// TwinCAT 3 PLC project mover_demo
// ProgramVersion: 3.1.4024.12
// libraries:
//   CmpBitmapPool, * (System)
//   Tc2_Standard, * (Beckhoff Automation GmbH)
//   Tc2_System, * (Beckhoff Automation GmbH)
//   Tc3_JsonXml, * (Beckhoff Automation GmbH)
//   Tc3_Module, * (Beckhoff Automation GmbH)
//   VisuDialogs, * (System)
// project tree:
//   DUTs/Helptec/ enLamp.TcDUT, enState.TcDUT, structAlarm.TcDUT, structButton.TcDUT
//   DUTs/ PieceType_e.TcTLEO, Mover_st.TcDUT, Piece_st.TcDUT
//   / GlobalTextList.TcGTLO, PlcTask.TcTTO, Visualization Manager.TcVMO (not stored), VISU_TASK.TcTTO (not stored)
//   GVLs/ CONST.TcGVL, GVL.TcGVL, HMI.TcGVL, IN.TcGVL, OUT.TcGVL, PERS.TcGVL, PRG.TcGVL, SIMU.TcGVL
//   POUs/00_MAIN/ MAIN.TcPOU, _05_FLAGS.TcPOU
//   POUs/10_HMI/FB%27s/ FB_BUTTON.TcPOU (not stored), FB_LampeBNI007F.TcPOU (not stored), FB_STATE.TcPOU (not stored)
//   POUs/10_HMI/ _10_HMI.TcPOU, _11_PAR_CHK.TcPOU, _14_STATE.TcPOU
//   POUs/20_AUTO/BuR SuperTrack com/ gMoverAxis.TcGVL, BR_PaletteCmd_t.TcDUT, BR_SectionCommand_t.TcDUT, PaletteCmd_bits_t.TcDUT, TC_to_BR_t.TcDUT, BR_to_TC_t.TcDUT, BR_TrackCommand_t.TcDUT
//   POUs/20_AUTO/FB%27s/ GetTick.TcPOU (not stored), getPercent.TcPOU (not stored)
//   POUs/20_AUTO/FB%27s/Vorlagen/ FB_ABL_VORLAGE.TcPOU (not stored), POU_AUT_VORLAGE.TcPOU (not stored), POU_ERR_VORLAGE.TcPOU (not stored), _01_MAIN.TcPOU (not stored)
//   POUs/20_AUTO/FileMan/ FB_FileMan.TcPOU, FB_ReadJSON.TcPOU, LoadFromMemory.TcPOU, SaveInMemory.TcPOU
//   POUs/20_AUTO/Mover/ ApproachScenario_e.TcTLEO, DistToTravel.TcPOU, FB_BasePieceHolder.TcPOU, FB_Group.TcPOU, FB_Mover.TcPOU, FB_MoverMan.TcPOU, FB_My_Piece.TcPOU, FB_Piece.TcPOU, FB_PieceHolderMover.TcPOU, FB_Position.TcPOU, FB_SimuMoverAxis.TcPOU, FB_SortMoverByPos.TcPOU, FB_PieceHolder.TcPOU, FB_StationMan.TcPOU, FB_Station.TcPOU, IProcessSampleMover.TcIO, ISimuMoverTimers.TcIO, IStation.TcIO, MoverDict.TcDUT, MoverDirection_e.TcTLEO, MoverState_e.TcTLEO, PiecePos_e.TcDUT, PieceState_e.TcDUT, Pos2D_t.TcDUT, ProcessExec_e.TcDUT, StationDict.TcDUT
//   POUs/20_AUTO/ST100/ F_GetPercent.TcPOU, ST100_Load_e.TcTLEO, FB_ABL_LOAD.TcPOU, FB_ABL_MODIFY.TcPOU, FB_ABL_UNLOAD.TcPOU, FB_AUT_ABSTRACT.TcPOU, FB_ABL_100.TcPOU, FB_AUT_LOAD.TcPOU, FB_AUT_MODIFY.TcPOU, FB_AUT_UNLOAD.TcPOU, ProcessExecution_e.TcTLEO, ST100_e.TcTLEO, ST100_Modify_e.TcTLEO, ST100_Unload_e.TcTLEO
//   POUs/20_AUTO/TOOL/ ASSERT.TcPOU, EqualApproximately.TcPOU, EqualDelta.TcPOU, EqualEssentially.TcPOU, IObject.TcIO, SortBubbleLREAL.TcPOU
//   POUs/20_AUTO/ _20_AUTO.TcPOU
//   VISUs/ Custom.TcIPO (not stored), VISU_main.TcVIS

CONFIGURATION mover_demo
    RESOURCE PLC ON TwinCAT3
        TASK PlcTask(INTERVAL := T#10ms, PRIORITY := 20);
        PROGRAM MAIN WITH PlcTask : MAIN;
        PROGRAM test WITH PlcTask : test;
    END_RESOURCE
END_CONFIGURATION

// ---- DUTs/Helptec/enLamp.TcDUT
{attribute 'qualified_only'}
{attribute 'strict'}
TYPE enLamp :
(
	Aus         := 2#0000,  //Aus
    Gruen       := 2#0001,  //Grün
    GruenB      := 2#1001,  //Grün blinkt
    Rot         := 2#0010,  //Rot
    RotB        := 2#1010,  //Rot blinkt
    Gelb        := 2#0011,  //Gelb
    GelbB       := 2#1011,  //Gelb blinkt
    Blau        := 2#0100,  //Blau 
    BlauB       := 2#1100,  //Blau blinkt
    Orange      := 2#0101,  //Orange
    OrangeB     := 2#1101,  //Orange blinkt
    Benutzer    := 2#0110,  //Benutzerdefiniert (Violet)
    BenutzerB   := 2#1110,  //Benutzerdefiniert blinkt (Violet)
    Weiss       := 2#0111,  //Weiss
    WeissB      := 2#1111   //Weiss blinkt
);
END_TYPE

// ---- DUTs/Helptec/enState.TcDUT
{attribute 'to_string'}
TYPE enState :
	//	MACHINE STATE
(
	StateOFF	,		(*0	OFF 		PLC STARTUP, EMERGENCY STOP	*)
	StateAIRon	,		(*1	AIR OK		AIRPRESSURE ON	 	*)
	StateENGIZED,		(*2	ENERGY OK	ENERGY/SECURITY CIRQUIT CLOSED	*)
	StateREF	,		(*3	HOMING		SYSTEM INITIAL RESET (HOMING AXIS ETC) *)
	StateMANU	,		(*4	MANUEL		MANUEL MODE (TEACH AXIS, MANEL MOVEMENT	*)
	StateINIT	,		(*5	INITIALISE	SYSTEM RESET 	*)
	StateREADY	,		(*6	READY		SYSTEM READY TO START	*)
	StateSTOP	,		(*7	STOP		SYSTEM STOPPED	*)
	StateALARM	,		(*8	ALARM		ALARM ACTIV	*)
	StateSTEP	,		(*9	STEP		STEP BY STEP MODE	*)
	StateEND	,		(*10 END		END MODE (FINISH ALL CYCLES	*)
	StateLEER	,		(*11 EMPTY		RUNNING TILL EMPTY STATE *)
	StateAUTO			(*12 RUN		RUNNING AUTOMATIC MODE	*)
);
END_TYPE

// ---- DUTs/Helptec/structAlarm.TcDUT
TYPE structAlarm :
STRUCT
	xAlarmIN	:	BOOL;	//Alarm Trigger
	xAlarmOFF	:	BOOL;	//Alarm übersteuert (wird nicht ausgelöst)
	xAlarmSAVE	:	BOOL;	//Alarm gespeichert (muss quittiert werden)
	xAlarmQUIT	:	BOOL;	//Alarm quittieren
	xAlarmOUT	:	BOOL;	//Alarm aktiv
	tAlarmVERZ	:	TIME;	//Alarmverzögerung
	sAlarmText	:	STRING;	//Alarmtext
	bAlarmNr	:	BYTE;	//Zusatztext #
END_STRUCT
END_TYPE

// ---- DUTs/Helptec/structButton.TcDUT
TYPE structButton :
STRUCT
	button	:	BOOL;	// BUTTON SIGNAL FROM HMI
	disable	:	BOOL;	// FORCE BUTTON INACTIV
	rtrig	:	BOOL;	// RISING EDGE
	ftrig	:	BOOL;	// FALLING EDGE
	press	:	BOOL;	// BUTTON PRESSED
	on		:	BOOL;	// FUNCTION ON (GREEN)
	error	:	BOOL;	// FUNCTION ERROR (RED)
END_STRUCT
END_TYPE

// ---- DUTs/PieceType_e.TcTLEO
{attribute 'qualified_only'}
{attribute 'strict'}
{attribute 'to_string'}
TYPE PieceType_e :
(
	long,
	short,
	_max
);
END_TYPE

// ---- DUTs/Mover_st.TcDUT
TYPE Mover_st :
STRUCT
	iStation	: INT;	// Number of the assigned station
	iPos		: INT;	// Current position
	pPiece		: POINTER TO Piece_st;	// Pointer to a pieces
END_STRUCT
END_TYPE

// ---- DUTs/Piece_st.TcDUT
TYPE Piece_st :
STRUCT
	iWorkingTimeMili	: INT;	// Time spent in a station, expressed in ms
	iWaitingTimeMili	: INT;	// Time spent out of any station, waiting to be proceed
	uiStartTimeMili		: UINT;	// Entering time in a station, expressed as task time
	UUID				: UDINT;	// Universal Unique ID
	eType				: PieceType_e;	// type of pieces
END_STRUCT
END_TYPE

// ---- POUs/20_AUTO/BuR SuperTrack com/BR_PaletteCmd_t.TcDUT
{attribute 'pack_mode=1'}
TYPE BR_PaletteCmd_t :
STRUCT
    cmd        : PaletteCmd_bits_t;
    nextTarget : USINT;
    offset     : ARRAY[0..2] OF USINT;
END_STRUCT
END_TYPE

// ---- POUs/20_AUTO/BuR SuperTrack com/BR_SectionCommand_t.TcDUT
{attribute 'pack_mode=1'}
TYPE BR_SectionCommand_t :
STRUCT
    enable : BIT;
END_STRUCT
END_TYPE

// ---- POUs/20_AUTO/BuR SuperTrack com/PaletteCmd_bits_t.TcDUT
TYPE PaletteCmd_bits_t :
STRUCT
    releaseToTargetOffset : BIT;
    direction             : BIT;
END_STRUCT
END_TYPE

// ---- POUs/20_AUTO/BuR SuperTrack com/TC_to_BR_t.TcDUT
{attribute 'pack_mode=1'}
TYPE TC_to_BR_t :
STRUCT
    trackCmd   : BR_TrackCommand_t;
    paletteNum : USINT;

    sectionCmd : BR_SectionCommand_t;

    missingPaletteIDs : ARRAY[0..20] OF USINT;

    palettesCmd : ARRAY[0..40] OF BR_PaletteCmd_t;

END_STRUCT
END_TYPE

// ---- POUs/20_AUTO/BuR SuperTrack com/BR_to_TC_t.TcDUT
{attribute 'pack_mode=1'}
TYPE BR_to_TC_t :
STRUCT
END_STRUCT
END_TYPE

// ---- POUs/20_AUTO/BuR SuperTrack com/BR_TrackCommand_t.TcDUT
{attribute 'pack_mode=1'}
TYPE BR_TrackCommand_t :
STRUCT
    enableAllSections        : BIT;
    releasePaletteAtTarget_1 : BIT;
    ApplyPaletteNumber       : BIT;
END_STRUCT
END_TYPE

// ---- POUs/20_AUTO/Mover/ApproachScenario_e.TcTLEO
{attribute 'qualified_only'}
{attribute 'strict'}
{attribute 'to_string'}
TYPE
ApproachScenario_e :
(
    WaitOnFinishedProcess,
    WaitOnFreeStation,
    DoNotWait,
    WaitOnPrevProcess,
    WaitOnExternalTrigger,
    _MAX
);
END_TYPE

// ---- POUs/20_AUTO/Mover/MoverDict.TcDUT
// Get information from a mover using this structure
TYPE MoverDict :
STRUCT
    MoverNum : INT;
    MoverPos : LREAL;
END_STRUCT
END_TYPE

// ---- POUs/20_AUTO/Mover/MoverDirection_e.TcTLEO
{attribute 'qualified_only'}
{attribute 'strict'}
TYPE MoverDirection_e :
(
	Farward,
	Reverse
);
END_TYPE

// ---- POUs/20_AUTO/Mover/MoverState_e.TcTLEO
{attribute 'qualified_only'}
{attribute 'strict'}
{attribute 'to_string'}
TYPE
MoverState_e :
(
    OperationDone,           // The operation on the mover is done, a new station needs to be given
    WaitOnNextStation,       // wait on the next station to be ready. The waiting depend on the scenario of the next station
    WaitLeaveCurrentStation, // If we are bind with the track system, we will be sure that we have actualy leaved the curent station
    MovingToStation,         // the mover is moving or try to move to the next station
    InStationPos,            // The mover is currently AT the station position (aka target pos.), waiting on the process TO begin
    InOperation,             // The attached process of the mover is running. The mover is not able to move
    PerformRelativeMove,     // Moving the mover when already in operation, go to WaitRelativeMoveEnd when mover actually moving
    WaitRelativeMoveEnd,     // Wait on the At_pos flag
    _MAX
);
END_TYPE

// ---- POUs/20_AUTO/Mover/PiecePos_e.TcDUT
{attribute 'qualified_only'}
{attribute 'strict'}
TYPE PiecePos_e :
(
    Assembly_left  := 0,
    Assembly_right := 1,
    Test_left      := 2,
    Test_right     := 3,
    _max           := 4
);
END_TYPE

// ---- POUs/20_AUTO/Mover/PieceState_e.TcDUT
{attribute 'qualified_only'}
{attribute 'strict'}
{attribute 'to_string'}
/// Piece status
TYPE PieceState_e :
(
    bad     := -1,
    good    := 0,
    working := 1 // a station works on a piece or has not finished its process
);
END_TYPE

// ---- POUs/20_AUTO/Mover/Pos2D_t.TcDUT
TYPE
Pos2D_t :
STRUCT
    x : DINT;
    y : DINT;
END_STRUCT
END_TYPE

// ---- POUs/20_AUTO/Mover/ProcessExec_e.TcDUT
{attribute 'qualified_only'}
{attribute 'strict'}
{attribute 'to_string'}
TYPE ProcessExec_e :
(
	StartImmediately,
	StartSynchronize,
	_MAX
);
END_TYPE

// ---- POUs/20_AUTO/Mover/StationDict.TcDUT
// Get information from a mover using this structure
TYPE StationDict :
STRUCT
    StationNum : INT;
    StationPos : LREAL;
END_STRUCT
END_TYPE

// ---- POUs/20_AUTO/ST100/ST100_Load_e.TcTLEO
{attribute 'qualified_only'}
{attribute 'strict'}
TYPE
ST100_Load_e :
(
    RESET := 0,         // Reset
    INIT := 100,        // Initialisieren 
    READY := 999,       // READY to Start, Init Done 
    START := 1000,      // Start Zyklisch
    MOVER_FREE_OP,      // Ab here, operation without mover can be done
    proceedOperation_1, // proceed to some operation
    waitOnMover,        // wait until the mover is there
    MOVER_NEEDED_OP,    // Ab here, a mover in position is needed to perform the action
    proceedOperation_2, // proceed to some operation
    SYNC_MOVER_LEAVE,   // MoverMan need to take the mover
    DONE := 8000,       // Ablauf beendet 
    ERROR := 9000,      // Fehler 
    _max
);
END_TYPE

// ---- POUs/20_AUTO/ST100/ProcessExecution_e.TcTLEO
{attribute 'qualified_only'}
{attribute 'strict'}
{attribute 'to_string'}
TYPE ProcessExecution_e :
(
	ExecuteImmediately,
	ExecuteWithPrevious,
	_MAX
);
END_TYPE

// ---- POUs/20_AUTO/ST100/ST100_e.TcTLEO
{attribute 'qualified_only'}
{attribute 'strict'}
{attribute 'to_string'}
TYPE
ST100_e :
(
    RESET := 0,         // Reset
    INIT := 100,        // Initialisieren 
    READY := 999,       // READY to Start, Init Done 
    START := 1000,      // Start Zyklisch
    MOVER_FREE_OP,      // Ab here, operation without mover can be done
    proceedOperation_1, //proceed to some operation
    waitOnMover,        // wait until the mover is there
    MOVER_NEEDED_OP,    // Ab here, a mover in position is needed to perform the action
    proceedOperation_2, //proceed to some operation
    DONE := 8000,       // Ablauf beendet 
    ERROR := 9000,      // Fehler 
    _max
);
END_TYPE

// ---- POUs/20_AUTO/ST100/ST100_Modify_e.TcTLEO
{attribute 'qualified_only'}
{attribute 'strict'}
TYPE ST100_Modify_e :
(
    RESET := 0,         // Reset
    INIT := 100,        // Initialisieren 
    READY := 999,       // READY to Start, Init Done 
    START := 1000,      // Start Zyklisch
    MOVER_FREE_OP,      // Ab here, operation without mover can be done
    waitOnMover,        // wait until the mover is there
    MOVER_NEEDED_OP,    // Ab here, a mover in position is needed to perform the action
    proceedOperation_1, //proceed to some operation
    proceedOperation_2, //proceed to some operation
    SYNC_MOVER_LEAVE,   // MoverMan need to take the mover
    DONE := 8000,       // Ablauf beendet 
    ERROR := 9000,      // Fehler 
    _max
);
END_TYPE

// ---- POUs/20_AUTO/ST100/ST100_Unload_e.TcTLEO
{attribute 'qualified_only'}
{attribute 'strict'}
TYPE ST100_Unload_e :
(
    RESET := 0,         // Reset
    INIT := 100,        // Initialisieren 
    READY := 999,       // READY to Start, Init Done 
    START := 1000,      // Start Zyklisch
    waitOnMover,        // wait until the mover is there
    MOVER_NEEDED_OP,    // Ab here, a mover in position is needed to perform the action
    proceedOperation_1, //proceed to some operation
    SYNC_MOVER_LEAVE,   // MoverMan need to take the mover
    MOVER_FREE_OP,      // Ab here, operation without mover can be done
    proceedOperation_2, //proceed to some operation
    DONE := 8000,       // Ablauf beendet 
    ERROR := 9000,      // Fehler 
    _max
);
END_TYPE

// ---- GVLs/CONST.TcGVL
{attribute 'qualified_only' := ''}
VAR_GLOBAL CONSTANT
    (*******************************************************************)
    (* Globale KONSTANTEN *)
    (*******************************************************************)

    USE_SIMULATION  : BOOL := TRUE;
    BIND_WITH_TRACK : BOOL := FALSE;

    STATION_NUMBER        : INT   := 18;
    MAX_GROUP             : INT   := 6;
    MAX_STATION_PER_GROUP : INT   := 8;
    RECIPE_NUMBER         : INT   := 4;
    MAX_TRACK_LENGTH      : LREAL := 10000;
    MAX_MOVER_SIZE        : LREAL := 200.0;

    MOVER_NUMBER : INT := 18;

    MAX_TRACK_OFFSET_LIST  : INT := 10;
    MAX_RECIPE_PER_STATION : INT := 10;
END_VAR

// ---- GVLs/GVL.TcGVL
{attribute 'qualified_only'}
VAR_GLOBAL
    (*******************************************************************)
    (* Allgemeine Globale Variablen *)
    (*******************************************************************)
    (******* FREIGABEN *********)
    //ST01
    xFG_ST01akVZ : BOOL; // Vereinzelung Teil anwesend
    xFG_ST01akWT : BOOL; // WT anwesend
    //ST02
    xFG_ST02akWT : BOOL; // WT anwesend

END_VAR

// ---- GVLs/HMI.TcGVL
{attribute 'qualified_only'}
VAR_GLOBAL
(*******************************************************************)
(* Globale HMI Variablen *)
(*******************************************************************)
	xImmer0	: 	BOOL := FALSE;	//ALLWAYS FALSE
	xImmer1	: 	BOOL := TRUE;	//ALLWAYS TRUE

(*******************************************************************)
(* Flags *)
(*******************************************************************)
	enState		:	enState;	//SYSTEM STATUS
	xInitDone	:	BOOL;		//SYSTEM INITIALIZED
	xRefDone	:	BOOL;		//Axis REF
	xAlarm		:	BOOL;		//ALARM AKTIV
	xMessage	:	BOOL;		//MELDUNG AKTIV
	xWait		:	BOOL;		//ALLE FBs warten
	xAIRon		:	BOOL;		//Luftdruck IO
	xSPC		:	BOOL;		//SPC angewählt

(*******************************************************************)
(* Buttons *)
(*******************************************************************)
	//Control
	btArMain	: ARRAY[0..20] OF structButton;	(*	
													0: AUTO
													1: STEP
													2: END
													3: MANU
													4: INIT
													5: STOP
													6: LEER
													7: QUIT
													8: RESET TEMP COUNTER
													9: START
													10: ...
												*)
	//Manuel Station 1
	btArManu01	: ARRAY[0..10] OF structButton;	(*	
													0: Zyklus	
													1: 101.01
													2: 101.02
													3: 101.03
													*)
	//Manuel Station 2
	btArManu02	: ARRAY[0..10] OF structButton;(*	
													0: Zyklus	
													1: 
													*)
	//Manuel Station 3
	btArManu03	: ARRAY[0..10] OF structButton;(*	
													0: Zyklus	
													1: 
													*)
	//Manuel Station 4
	btArManu04	: ARRAY[0..10] OF structButton;	(*	
													0: Zyklus	
													1: 
													*)
	//Manuel Station 5
	btArManu05	: ARRAY[0..10] OF structButton;(*	
													0: Zyklus	
													1: 
													*)
	//Manuel Station 6
	btArManu06	: ARRAY[0..10] OF structButton;(*	
													0: Zyklus	
													1: 
													*)
	//Manuel Station 7
	btArManu07	: ARRAY[0..10] OF structButton;(*	
													0: Zyklus	
													1: 
													*)
	//Manuel Station 8
	btArManu08	: ARRAY[0..10] OF structButton;(*	
													0: Zyklus	
													1: 
													*)
	//Manuel Station 9
	btArManu09	: ARRAY[0..10] OF structButton;(*	
													0: Zyklus	
													1: 
													*)
	//Manuel Station 10
	btArManu10	: ARRAY[0..10] OF structButton;(*	
													0: Zyklus	
													1: 
													*) 

(*******************************************************************)
(* ALARME  *)
(*******************************************************************)				
	strArALARM : ARRAY [1..100] OF structAlarm;	
	strArMSG : ARRAY [1..100] OF structAlarm;
	xArAlarmHMI : ARRAY [1..9999] OF BOOL;
	
(*******************************************************************)
(* ANZEIGE - Werte *)
(*******************************************************************)

(*******************************************************************)
(* Cycle Time [STATION]*)
(*******************************************************************)
	dwArStartTime	: 	ARRAY[0..10] OF DWORD;
	dwArCycleTime	: 	ARRAY[0..10] OF DWORD;
	
(*******************************************************************)
(* Diverses *)
(*******************************************************************)
	xWriteALlog: BOOL;	//Alarmlog schreiben in File
END_VAR

// ---- GVLs/IN.TcGVL
{attribute 'qualified_only'}
VAR_GLOBAL
(*******************************************************************)
(* EINGÄNGE *)
(*******************************************************************)
	(* Modul *)
	//-EL#
//	I000_24VDC			AT %IX0.0		:	BOOL;			//Überwachung +24VDC
//	I001_				AT %IX0.1		:	BOOL;			//
//	I002_				AT %IX0.2		:	BOOL;			//    
//	I003_		    	AT %IX0.3		:	BOOL;			//	
//	I004_				AT %IX0.4		:	BOOL;			//Reserve
//	I005_				AT %IX0.5		:	BOOL;			//Reserve
//	I006_				AT %IX0.6		:	BOOL;			//Reserve    
//	I007_				AT %IX0.7		:	BOOL;			//Reserve
//	
//	I010_				AT %IX1.0		:	BOOL;			//Taktsignal Presse
//	I011_				AT %IX1.1		:	BOOL;			//Presse Bereit
//	I012_				AT %IX1.2		:	BOOL;			//Reserve Presse
//	I013_				AT %IX1.3		:	BOOL;			//Reserve Presse
//	I014_				AT %IX1.4		:	BOOL;			//Reserve
//	I015_				AT %IX1.5		:	BOOL;			//Reserve
//	I016_				AT %IX1.6		:	BOOL;			//Reserve
//	I017_				AT %IX1.7		:	BOOL;			//Reserve
//	
//	
//	(* IO-Link Boxen *)
//(*******************************************************************)
//	//-5001
//	(*Beispiel 	ST01 	Stopper Mono (nur GS), Greifer Mono, 
//						Vereinzelung Bi, AK WT, AK Teil, STAU WF
//	*)
//	IB5001				AT %IB5001			:	BYTE;			//Input Byte Box 1
//	I101_01_GS			AT %IX5001.0		:	BOOL;			//Stopper GS
//	I101_02_UH			AT %IX5001.1		:	BOOL;			//Greifer GS
//	I101_02_AS			AT %IX5001.2		:	BOOL;			//Greifer AS
//	I101_03_GS			AT %IX5001.3		:	BOOL;			//Vereinzelung GS
//	I101_03_AS			AT %IX5001.4		:	BOOL;			//Vereinzelung AS
//	I101_WT				AT %IX5001.5		:	BOOL;			//AK WT	
//	I101_AK				AT %IX5001.6		:	BOOL;			//AK Teil
//	I101_STAU			AT %IX5001.7		:	BOOL;			//Stau Zuführung
//	
//	//-5002
//	(*Beispiel 	ST02 	Stopper Mono (nur GS), Indexierer Mono, 
//						Presse Mono, AK WT, AK Teil
//	*)
//	IB5002				AT %IB5002			:	BYTE;			//Input Byte Box 2
//	I102_01_GS			AT %IX5002.0		:	BOOL;			//Stopper GS
//	I102_02_GS			AT %IX5002.1		:	BOOL;			//Index GS
//	I102_02_AS			AT %IX5002.2		:	BOOL;			//Index AS
//	I102_03_GS			AT %IX5002.3		:	BOOL;			//Pressen GS
//	I102_03_AS			AT %IX5002.4		:	BOOL;			//Pressen AS
//	I102_WT				AT %IX5002.5		:	BOOL;			//AK WT	
//	I102_AK				AT %IX5002.6		:	BOOL;			//AK Teil
//	I102_STAU			AT %IX5002.7		:	BOOL;			//
//	(*
//	IB5001				AT %IB5001			:	BYTE;			//Input Byte Box 1
//	I5001_0_			AT %IX5001.0		:	BOOL;			//
//	I5001_1_			AT %IX5001.1		:	BOOL;			//
//	I5001_2_			AT %IX5001.2		:	BOOL;			//
//	I5001_3_			AT %IX5001.3		:	BOOL;			//
//	I5001_4_			AT %IX5001.4		:	BOOL;			//
//	I5001_5_			AT %IX5001.5		:	BOOL;			//	
//	I5001_6_			AT %IX5001.6		:	BOOL;			//
//	I5001_7_			AT %IX5001.7		:	BOOL;			//
//	
//	//-5002
//	IB5002				AT %IB5002			:	BYTE;			//Input Byte Box 2
//	I5002_0_			AT %IX5002.0		:	BOOL;			//
//	I5002_1_			AT %IX5002.1		:	BOOL;			//
//	I5002_2_			AT %IX5002.2		:	BOOL;			//
//	I5002_3_			AT %IX5002.3		:	BOOL;			//
//	I5002_4_			AT %IX5002.4		:	BOOL;			//
//	I5002_5_			AT %IX5002.5		:	BOOL;			//	
//	I5002_6_			AT %IX5002.6		:	BOOL;			//
//	I5002_7_			AT %IX5002.7		:	BOOL;			//
//	*)
//	//-5003
//	IB5003				AT %IB5003			:	BYTE;			//Input Byte Box 3
//	I5003_0_			AT %IX5003.0		:	BOOL;			//
//	I5003_1_			AT %IX5003.1		:	BOOL;			//
//	I5003_2_			AT %IX5003.2		:	BOOL;			//
//	I5003_3_			AT %IX5003.3		:	BOOL;			//
//	I5003_4_			AT %IX5003.4		:	BOOL;			//
//	I5003_5_			AT %IX5003.5		:	BOOL;			//	
//	I5003_6_			AT %IX5003.6		:	BOOL;			//
//	I5003_7_			AT %IX5003.7		:	BOOL;			//
//	
//	//-5004
//	IB5004				AT %IB5004			:	BYTE;			//Input Byte Box 4
//	I5004_0_			AT %IX5004.0		:	BOOL;			//
//	I5004_1_			AT %IX5004.1		:	BOOL;			//
//	I5004_2_			AT %IX5004.2		:	BOOL;			//
//	I5004_3_			AT %IX5004.3		:	BOOL;			//
//	I5004_4_			AT %IX5004.4		:	BOOL;			//
//	I5004_5_			AT %IX5004.5		:	BOOL;			//	
//	I5004_6_			AT %IX5004.6		:	BOOL;			//
//	I5004_7_			AT %IX5004.7		:	BOOL;			//
//	
//	//-5005
//	IB5005				AT %IB5005			:	BYTE;			//Input Byte Box 5
//	I5005_0_			AT %IX5005.0		:	BOOL;			//
//	I5005_1_			AT %IX5005.1		:	BOOL;			//
//	I5005_2_			AT %IX5005.2		:	BOOL;			//
//	I5005_3_			AT %IX5005.3		:	BOOL;			//
//	I5005_4_			AT %IX5005.4		:	BOOL;			//
//	I5005_5_			AT %IX5005.5		:	BOOL;			//	
//	I5005_6_			AT %IX5005.6		:	BOOL;			//
//	I5005_7_			AT %IX5005.7		:	BOOL;			//
//	
//	//-5006
//	IB5006				AT %IB5006			:	BYTE;			//Input Byte Box 6
//	I5006_0_			AT %IX5006.0		:	BOOL;			//
//	I5006_1_			AT %IX5006.1		:	BOOL;			//
//	I5006_2_			AT %IX5006.2		:	BOOL;			//
//	I5006_3_			AT %IX5006.3		:	BOOL;			//
//	I5006_4_			AT %IX5006.4		:	BOOL;			//
//	I5006_5_			AT %IX5006.5		:	BOOL;			//	
//	I5006_6_			AT %IX5006.6		:	BOOL;			//
//	I5006_7_			AT %IX5006.7		:	BOOL;			//
//	
//	//-5007
//	IB5007				AT %IB5007			:	BYTE;			//Input Byte Box 7
//	I5007_0_			AT %IX5007.0		:	BOOL;			//
//	I5007_1_			AT %IX5007.1		:	BOOL;			//
//	I5007_2_			AT %IX5007.2		:	BOOL;			//
//	I5007_3_			AT %IX5007.3		:	BOOL;			//
//	I5007_4_			AT %IX5007.4		:	BOOL;			//
//	I5007_5_			AT %IX5007.5		:	BOOL;			//	
//	I5007_6_			AT %IX5007.6		:	BOOL;			//
//	I5007_7_			AT %IX5007.7		:	BOOL;			//
//	
//	//-5008
//	IB5008				AT %IB5008			:	BYTE;			//Input Byte Box 8
//	I5008_0_			AT %IX5008.0		:	BOOL;			//
//	I5008_1_			AT %IX5008.1		:	BOOL;			//
//	I5008_2_			AT %IX5008.2		:	BOOL;			//
//	I5008_3_			AT %IX5008.3		:	BOOL;			//
//	I5008_4_			AT %IX5008.4		:	BOOL;			//
//	I5008_5_			AT %IX5008.5		:	BOOL;			//	
//	I5008_6_			AT %IX5008.6		:	BOOL;			//
//	I5008_7_			AT %IX5008.7		:	BOOL;			//
//	
//	//-5009
//	IB5009				AT %IB5009			:	BYTE;			//Input Byte Box 9
//	I5009_0_			AT %IX5009.0		:	BOOL;			//
//	I5009_1_			AT %IX5009.1		:	BOOL;			//
//	I5009_2_			AT %IX5009.2		:	BOOL;			//
//	I5009_3_			AT %IX5009.3		:	BOOL;			//
//	I5009_4_			AT %IX5009.4		:	BOOL;			//
//	I5009_5_			AT %IX5009.5		:	BOOL;			//	
//	I5009_6_			AT %IX5009.6		:	BOOL;			//
//	I5009_7_			AT %IX5009.7		:	BOOL;			//
//	
//	//-5010
//	IB5010				AT %IB5010			:	BYTE;			//Input Byte Box 10
//	I5010_0_			AT %IX5010.0		:	BOOL;			//
//	I5010_1_			AT %IX5010.1		:	BOOL;			//
//	I5010_2_			AT %IX5010.2		:	BOOL;			//
//	I5010_3_			AT %IX5010.3		:	BOOL;			//
//	I5010_4_			AT %IX5010.4		:	BOOL;			//
//	I5010_5_			AT %IX5010.5		:	BOOL;			//	
//	I5010_6_			AT %IX5010.6		:	BOOL;			//
//	I5010_7_			AT %IX5010.7		:	BOOL;			//
	
END_VAR

// ---- GVLs/OUT.TcGVL
{attribute 'qualified_only'}
VAR_GLOBAL
(*******************************************************************)
(* AUSGÄNGE *)
(*******************************************************************)
	(* Modul *)	
	//-EL#
//	Q000_LAMP_NRJ		AT %QX0.0		:	BOOL;			//Lampe Energie
//	Q001_TuerVer		AT %QX0.1		:	BOOL;			//Türen verriegelt
//	Q002_				AT %QX0.2		:	BOOL;			//
//	Q003_				AT %QX0.3		:	BOOL;			//Reserve
//	Q004_WF_FG			AT %QX0.4		:	BOOL;			//ST01 Freigabe WF 
//	Q005_				AT %QX0.5		:	BOOL;			//Reserve
//	Q006_				AT %QX0.6		:	BOOL;			//
//	Q007_				AT %QX0.7		:	BOOL;			//
//	
//	Q010_				AT %QX1.0		:	BOOL;			//
//	Q011_				AT %QX1.1		:	BOOL;			//
//	Q012_				AT %QX1.2		:	BOOL;			//Reserve
//	Q013_				AT %QX1.3		:	BOOL;			//Reserve
//	Q014_				AT %QX1.4		:	BOOL;			//Reserve
//	Q015_				AT %QX1.5		:	BOOL;			//Reserve
//	Q016_				AT %QX1.6		:	BOOL;			//Reserve
//	Q017_				AT %QX1.7		:	BOOL;			//Reserve
//			
//
//	(* IO-Link  *)
//(*******************************************************************)
//	(* Lampe *)
//	QW194A3				AT%Q*			:	WORD;			//Signallampe1
//	QW194A6				AT%Q*			: 	WORD;			//Signallampe2
//	
//	Q194A3_SycStart		AT %Q*			:	BOOL;			//Syscstart 194A3
//	Q194A6_SycStart		AT %Q*			:	BOOL;			//Syscstart 194A6	
//	Q194A3_SycImp		AT %Q*			:	BOOL;			//SyscImp 194A3
//	Q194A6_SycImp		AT %Q*			:	BOOL;			//SyscImp 194A6		
//	
//	(* Boxen *)
//	(*Beispiel 	ST01 Stopper Mono, Greifer Mono, Vereinzelung Bi,
//				ST02 Stopper Mono, Indexierer Mono, Presse Mono
//	*)
//	Q101_01_AS			AT	%QX2000.0	:	BOOL;			//101.01 Stopper
//	Q200A1_1_12			AT	%QX2000.1	:	BOOL;			//
//	Q101_02_AS			AT	%QX2000.2	:	BOOL;			//101.02 Greifer
//	Q200A1_2_12			AT	%QX2000.3	:	BOOL;			//
//	Q101_03_AS			AT	%QX2000.4	:	BOOL;			//101.03 Vereinzelung AS
//	Q101_03_GS			AT	%QX2000.5	:	BOOL;			//101.03 Vereinzelung GS
//	Q102_01_AS			AT	%QX2000.6	:	BOOL;			//102.01 Stopper
//	Q200A1_4_12			AT	%QX2000.7	:	BOOL;			//
//	Q102_02_AS			AT	%QX2000.8	:	BOOL;			//102.02 Indexieren
//	Q200A1_5_12			AT	%QX2000.9	:	BOOL;			//
//	Q102_03_AS			AT	%QX2000.10	:	BOOL;			//102.03 Pressen
//	Q200A1_6_12			AT	%QX2000.11	:	BOOL;			//
//	Q200A1_7_14			AT	%QX2000.12	:	BOOL;			//
//	Q200A1_7_12			AT	%QX2000.13	:	BOOL;			//
//	Q200A1_8_14			AT	%QX2000.14	:	BOOL;			//
//	Q200A1_8_12			AT	%QX2000.15	:	BOOL;			//
//(*	QW200A1				AT	%QB2000		:	WORD;			//IO-Link 8er VENTILBLOCK 
//	Q200A1_1_14			AT	%QX2000.0	:	BOOL;			//
//	Q200A1_1_12			AT	%QX2000.1	:	BOOL;			//
//	Q200A1_2_14			AT	%QX2000.2	:	BOOL;			//
//	Q200A1_2_12			AT	%QX2000.3	:	BOOL;			//
//	Q200A1_3_14			AT	%QX2000.4	:	BOOL;			//
//	Q200A1_3_12			AT	%QX2000.5	:	BOOL;			//
//	Q200A1_4_14			AT	%QX2000.6	:	BOOL;			//
//	Q200A1_4_12			AT	%QX2000.7	:	BOOL;			//
//	Q200A1_5_14			AT	%QX2000.8	:	BOOL;			//
//	Q200A1_5_12			AT	%QX2000.9	:	BOOL;			//
//	Q200A1_6_14			AT	%QX2000.10	:	BOOL;			//
//	Q200A1_6_12			AT	%QX2000.11	:	BOOL;			//
//	Q200A1_7_14			AT	%QX2000.12	:	BOOL;			//
//	Q200A1_7_12			AT	%QX2000.13	:	BOOL;			//
//	Q200A1_8_14			AT	%QX2000.14	:	BOOL;			//
//	Q200A1_8_12			AT	%QX2000.15	:	BOOL;			//
//*)	
//	QW200A2				AT	%QB2002		:	WORD;			//IO-Link 8er VENTILBLOCK 
//	Q200A2_1_14			AT	%QX2002.0	:	BOOL;			//
//	Q200A2_1_12			AT	%QX2002.1	:	BOOL;			//
//	Q200A2_2_14			AT	%QX2002.2	:	BOOL;			//
//	Q200A2_2_12			AT	%QX2002.3	:	BOOL;			//
//	Q200A2_3_14			AT	%QX2002.4	:	BOOL;			//
//	Q200A2_3_12			AT	%QX2002.5	:	BOOL;			//
//	Q200A2_4_14			AT	%QX2002.6	:	BOOL;			//
//	Q200A2_4_12			AT	%QX2002.7	:	BOOL;			//
//	Q200A2_5_14			AT	%QX2002.8	:	BOOL;			//
//	Q200A2_5_12			AT	%QX2002.9	:	BOOL;			//
//	Q200A2_6_14			AT	%QX2002.10	:	BOOL;			//
//	Q200A2_6_12			AT	%QX2002.11	:	BOOL;			//
//	Q200A2_7_14			AT	%QX2002.12	:	BOOL;			//
//	Q200A2_7_12			AT	%QX2002.13	:	BOOL;			//
//	Q200A2_8_14			AT	%QX2002.14	:	BOOL;			//
//	Q200A2_8_12			AT	%QX2002.15	:	BOOL;			//


	
END_VAR

// ---- GVLs/PERS.TcGVL
{attribute 'qualified_only'}
VAR_GLOBAL RETAIN
    (***********************************************************************************************)
    (* COUNTER *)
    (***********************************************************************************************)
    //COUNTER 
    udiTotalOK  : UDINT; // Total Counter  OK 
    udiTotalNOK : UDINT; // Total Counter  NOK 

    udiTempOK  : UDINT; // Temporary Counter  OK 
    udiTempNOK : UDINT; // Temporary Counter  NOK 

    //OPERATING HOURS
    udiCountHon    : UDINT; // Operating hours SYSTEM POWER ON [h] 
    udiCount6Mon   : UDINT; // Operating hours SYSTEM POWER ON [6min (0.1h)] 
    udiCountHauto  : UDINT; // Operating hours SYSTEM IN AUTOMATIC MODE [h] 
    udiCount6Mauto : UDINT; // Operating hours SYSTEM IN AUTOMATIC MODE [6min (0.1h)] 

    (***********************************************************************************************)
    (* Application *)
    (***********************************************************************************************)
    iStationTimeDef1 : ARRAY[1..CONST.STATION_NUMBER] OF DINT;
    iStationTimeDef2 : ARRAY[1..CONST.STATION_NUMBER] OF DINT;

    iRecipeCurrent : INT;
    arrStationOffsetsList : ARRAY[0..CONST.MAX_TRACK_OFFSET_LIST - 1] OF ARRAY[1..CONST.STATION_NUMBER] OF REAL;
    arrStationUsedList : ARRAY[0..CONST.MAX_RECIPE_PER_STATION - 1] OF ARRAY[1..CONST.STATION_NUMBER] OF INT;

END_VAR

// ---- GVLs/PRG.TcGVL
{attribute 'qualified_only'}
VAR_GLOBAL
    st105_aut  : FB_AUT_LOAD;   // Laden Filtergehäuse
    st110_aut  : FB_AUT_LOAD;   // Laden RFID-Ring
    st115_aut  : FB_AUT_LOAD;   // Laden kristal
    st120_aut  : FB_AUT_LOAD;   // Laden Solerohr
    st125_aut  : FB_AUT_LOAD;   // Laden filterhut
    st130_aut  : FB_AUT_MODIFY; // Dosieren A
    st135_aut  : FB_AUT_MODIFY; // Dosieren B
    st140_aut  : FB_AUT_MODIFY; // Niveaukontrolle
    st145_aut  : FB_AUT_LOAD;   // Laden Patronendeckel
    st150_aut : FB_AUT_MODIFY; // Utralson A
    st155_aut : FB_AUT_MODIFY; // Ultrason B
    st160_aut : FB_AUT_MODIFY; // Prüfig A
    st165_aut : FB_AUT_MODIFY; // Prüfig B
    st170_aut : FB_AUT_MODIFY; // Program RFID
    st175_aut : FB_AUT_MODIFY; // Laser A
    st176_aut : FB_AUT_MODIFY; // Laser B
    st180_aut : FB_AUT_UNLOAD; // Entladen schlecht
    st185_aut : FB_AUT_UNLOAD; // Entladen gut
END_VAR

// ---- GVLs/SIMU.TcGVL
{attribute 'qualified_only'}
VAR_GLOBAL
    iCompletionHMI : ARRAY[0..CONST.STATION_NUMBER] OF INT;

    lrSpeedMover       : LREAL := 20.0;
    lrAccelMover       : LREAL; // is lrAccelMoverSlider^2
    lrAccelMoverSlider : LREAL := 0.4;
END_VAR

// ---- POUs/20_AUTO/BuR SuperTrack com/gMoverAxis.TcGVL
{attribute 'qualified_only'}
VAR_GLOBAL
    I_CT_Shuttle_from_BR AT %I* : CT_Shuttle_BR_to_Tc_u; // all the movers
    Q_CT_Shuttle_to_BR   AT %Q* : CT_Shuttle_Tc_to_BR_u;
    I_CT_Track_from_BR   AT %I* : CT_Track_BR_to_Tc_u;
    Q_CT_Track_to_BR     AT %Q* : CT_Track_Tc_to_BR_u;

END_VAR

// ---- POUs/20_AUTO/Mover/IProcessSampleMover.TcIO
INTERFACE IProcessSampleMover

METHOD GiveMover : IProcessSampleMover
VAR_INPUT
	mover : REFERENCE TO FB_Mover;
END_VAR
END_METHOD

(* % of completion of the process *)
PROPERTY iCompletionPC : INT
GET
END_GET
END_PROPERTY

PROPERTY Mover : REFERENCE TO FB_Mover
GET
END_GET
SET
END_SET
END_PROPERTY

PROPERTY ProcessExecution : ProcessExecution_e
GET
END_GET
SET
END_SET
END_PROPERTY

METHOD TakeMover : IProcessSampleMover
VAR_INPUT
END_VAR
END_METHOD

METHOD ToString : STRING
VAR_INPUT
END_VAR
END_METHOD

PROPERTY xBusy : BOOL
GET
END_GET
SET
END_SET
END_PROPERTY

PROPERTY xDone : BOOL
GET
END_GET
END_PROPERTY

PROPERTY xMoverPathFree : BOOL
GET
END_GET
END_PROPERTY

PROPERTY xMoverShouldLeave : BOOL
GET
END_GET
END_PROPERTY

END_INTERFACE

// ---- POUs/20_AUTO/Mover/ISimuMoverTimers.TcIO
INTERFACE ISimuMoverTimers

(* Process time, expressed in milisecond *)
PROPERTY iProcessTimeMili_1 : DINT
GET
END_GET
SET
END_SET
END_PROPERTY

(* Process time, expressed in milisecond *)
PROPERTY iProcessTimeMili_2 : DINT
GET
END_GET
SET
END_SET
END_PROPERTY

END_INTERFACE

// ---- POUs/20_AUTO/Mover/IStation.TcIO
INTERFACE IStation

PROPERTY Position : REFERENCE TO FB_Position
GET
END_GET
SET
END_SET
END_PROPERTY

PROPERTY Process : REFERENCE TO FB_AUT_ABSTRACT
GET
END_GET
SET
END_SET
END_PROPERTY

END_INTERFACE

// ---- POUs/20_AUTO/TOOL/IObject.TcIO
// Basic object interface that provide core function for each FB
INTERFACE IObject

METHOD Equals : BOOL
VAR_INPUT
	object : ANY;
END_VAR
END_METHOD

METHOD ToString : STRING
VAR_INPUT
END_VAR
END_METHOD

END_INTERFACE

// ---- POUs/00_MAIN/MAIN.TcPOU
PROGRAM MAIN
VAR
	MoverMan	: FB_MoverMan;
END_VAR


_05_FLAGS( xIN_AIR:=TRUE, xIN_btRES_TEMP:=HMI.btArMain[8]);

//HMI
_10_HMI();

MoverMan();

//AUTO
_20_AUTO(xIN_Quit:= _14_STATE._FB_btQUIT.pbtIN^.rtrig , enIN_State:= HMI.enState);

END_PROGRAM

// ---- POUs/20_AUTO/Mover/FB_MoverMan.TcPOU
FUNCTION_BLOCK FB_MoverMan
VAR_INPUT
END_VAR
VAR_OUTPUT
    xOUT_AllMoverEmpty : BOOL; // TRUE when LastStationVisited from all shuttle are 0
    xOUT_Error         : BOOL; // CleverTrack is in error and needs a reset
END_VAR
VAR
    {attribute 'no_copy'}
    _PieceHolderList : ARRAY[1..2] OF FB_PieceHolderMover[
        (0),
        (0)];

    {attribute 'no_copy'}
    _SimuMoverList : ARRAY[1..19] OF FB_SimuMoverAxis[
        (116),
        (433),
        (750),
        (1067),
        (1384),
        (1701),
        (2018),
        (2335),
        (2652),
        (3000),
        (3400),
        (3800),
        (5200),
        (5600),
        (6000),
        (6400),
        (6800),
        (7200),
        (7600)];

    {attribute 'no_copy'}
    _MoverList : ARRAY[1..19] OF FB_Mover[
        (1, _SimuMoverList[1]),
        (2, _SimuMoverList[2]),
        (3, _SimuMoverList[3]),
        (4, _SimuMoverList[4]),
        (5, _SimuMoverList[5]),
        (6, _SimuMoverList[6]),
        (7, _SimuMoverList[7]),
        (8, _SimuMoverList[8]),
        (9, _SimuMoverList[9]),
        (10, _SimuMoverList[10]),
        (11, _SimuMoverList[11]),
        (12, _SimuMoverList[12]),
        (13, _SimuMoverList[13]),
        (14, _SimuMoverList[14]),
        (15, _SimuMoverList[15]),
        (16, _SimuMoverList[16]),
        (17, _SimuMoverList[17]),
        (18, _SimuMoverList[18]),
        (19, _SimuMoverList[19])];

    {attribute 'no_copy'}
    _PosList : ARRAY[1..CONST.STATION_NUMBER] OF FB_Position[
        (125, 1, 1),  // 105
        (625, 1, 1),  // 110
        (1125, 1, 1), // 115
        (1375, 1, 1), // 120
        (1625, 1, 1), // 125
        (2375, 1, 1), // 130
        (2625, 1, 1), // 135
        (2875, 1, 1), // 140
        (3125, 1, 1), // 145
        (3625, 1, 1), // 150
        (3875, 1, 1), // 155
        // second part
        (5205, 1, 1), // 160
        (5455, 1, 1), // 165
        (5897, 1, 1), // 170
        (7365, 1, 1), // 175
        (7630, 1, 1), // 176
        (8655, 1, 1), // 180
        (8905, 1, 1)  // 185
    ];

    {attribute 'no_copy'}
    _StationList : ARRAY[1..CONST.STATION_NUMBER] OF
        FB_Station[
        (_PosList[1],
         PRG.st105_aut,
         0,
         ApproachScenario_e.DoNotWait,
         3,
         5),
        (_PosList[2],
         PRG.st110_aut,
         0,
         ApproachScenario_e.DoNotWait,
         3,
         10),
        (_PosList[3],
         PRG.st115_aut,
         0,
         ApproachScenario_e.DoNotWait,
         3,
         15),
        (_PosList[4],
         PRG.st120_aut,
         0,
         ApproachScenario_e.DoNotWait,
         3,
         20),
        (_PosList[6],
         PRG.st125_aut,
         0,
         ApproachScenario_e.DoNotWait,
         3,
         25),
        (_PosList[5],
         PRG.st130_aut,
         0,
         ApproachScenario_e.DoNotWait,
         3,
         30),
        (_PosList[7],
         PRG.st135_aut,
         0,
         ApproachScenario_e.DoNotWait,
         3,
         35),
        (_PosList[8],
         PRG.st140_aut,
         0,
         ApproachScenario_e.DoNotWait,
         3,
         40),
        (_PosList[9],
         PRG.st145_aut,
         0,
         ApproachScenario_e.DoNotWait,
         3,
         45),
        (_PosList[10],
         PRG.st150_aut,
         0,
         ApproachScenario_e.DoNotWait,
         3,
         50),
        (_PosList[11],
         PRG.st155_aut,
         0,
         ApproachScenario_e.DoNotWait,
         3,
         55),
        (_PosList[12],
         PRG.st160_aut,
         0,
         ApproachScenario_e.DoNotWait,
         3,
         60),
        (_PosList[13],
         PRG.st165_aut,
         0,
         ApproachScenario_e.DoNotWait,
         3,
         65),
        (_PosList[14],
         PRG.st170_aut,
         0,
         ApproachScenario_e.DoNotWait,
         3,
         70),
        (_PosList[15],
         PRG.st175_aut,
         0,
         ApproachScenario_e.DoNotWait,
         3,
         75),
        (_PosList[16],
         PRG.st176_aut,
         0,
         ApproachScenario_e.DoNotWait,
         3,
         76),
        (_PosList[17],
         PRG.st180_aut,
         0,
         ApproachScenario_e.DoNotWait,
         3,
         80),
        (_PosList[18],
         PRG.st185_aut,
         0,
         ApproachScenario_e.DoNotWait,
         3,
         85)];

    // Smart
    {attribute 'no_copy'}
    _StationSet1 :
        ARRAY[1..CONST.STATION_NUMBER] OF INT := [0,  // ST105
                                                  0,  // ST110
                                                  -1, // ST115
                                                  0,  // ST120
                                                  0,  // ST125
                                                  0,  // ST130
                                                  0,  // ST135
                                                  0,  // ST140
                                                  0,  // ST145
                                                  0,  // ST150
                                                  0,  // ST155
                                                  0,  // ST160
                                                  0,  // ST165
                                                  0,  // ST170
                                                  1,  // ST175
                                                  1,  // ST176
                                                  0,  // ST180
                                                  0]; // ST185

    {attribute 'no_copy'}
    _SelWorkStationList : ARRAY[1..7] OF POINTER TO ARRAY[1..CONST.STATION_NUMBER] OF INT
        := [ADR(_StationSet1),
            ADR(_StationSet1),
            ADR(_StationSet1),
            ADR(_StationSet1),
            ADR(_StationSet1),
            ADR(_StationSet1),
            ADR(_StationSet1)];

    {attribute 'no_copy'}
    _WorkStationList : FB_StationMan(
        ADR(_StationList),
        ADR(PERS.arrStationUsedList),
        _PieceHolderList[1]);

    step : INT := 0; //test step

    mv_i                : INT;           // mover index
    bMoverSync          : BOOL := FALSE; // external trigger for movers
    iNumOfMoverOnTheWay : INT;           // temp var to know how many mover there are between a given mover and its next station

    lastEmptyStation : REFERENCE TO FB_Station; // temp var to store the next free station
    tempMover        : REFERENCE TO FB_Mover;

    HMI_Scenario   : ApproachScenario_e := ApproachScenario_e.WaitOnFinishedProcess;
    HMI_TimeAvg    : DINT               := 1000;
    HMI_TimeMin    : DINT               := 900;
    HMI_TimeMax    : DINT               := 1100;
    HMI_xStopMover : BOOL               := FALSE;
    HMI_iSelMover  : INT                := 1;

    HMI_Bp_Enable_Power   : structButton;
    fb_Bp_Enable_Power    : FB_BUTTON;
    HMI_Bp_Enable_Process : structButton;
    fb_Bp_Enable_Process  : FB_BUTTON;

    HMI_send_all_shuttle_to_unload : BOOL;

    RT_apply_station_list : Tc2_Standard.R_TRIG;

    old_recipe : INT;

    _iID : INT := 0; // instance ID, is set during FB_Init using the value of _iInstanceCounter 
END_VAR
VAR CONSTANT
    TRACK_SIMULATION : BOOL := FALSE; // Set to true when supertrack is in simulation
END_VAR
VAR_STAT
    _iInstanceCounter : INT := 1; // instance counter
END_VAR

(* ---------------------------------------------------------------------------- *)
(* THIS IS A PARTICULAR IMPLEMENTATION OF CLEVERTRAKLIB. THIS SHOULD BE REMOVED *)
CASE step OF

0: // setup everything
    FOR mv_i := 1 TO CONST.MOVER_NUMBER BY 1 DO
        _MoverList[mv_i].SetStation(_WorkStationList.GetStartStation(_MoverList[mv_i].MoverAxis.CurrentPos)^);
        // _MoverList[mv_i].SetPieceHolder( _WorkStationList[PH_num].PieceHolder);
    END_FOR

    step := 5;

5: // wait until the whole path is free
    IF gMoverAxis.Q_CT_Track_to_BR.asStruct.bCommand.wholePathFree AND
       (HMI.enState <> enState.StateMANU) THEN
        step := 10;
    ELSIF NOT CONST.BIND_WITH_TRACK THEN
        step := 15;
    END_IF

10: // turn power on
    gMoverAxis.Q_CT_Track_to_BR.asStruct.bCommand.enablePower := (HMI.enState <> enState.StateMANU);

    IF gMoverAxis.I_CT_Track_from_BR.asStruct.bStatus.powerOn THEN

        FOR mv_i := 1 TO CONST.MOVER_NUMBER - 1 BY 1 DO
            gMoverAxis.Q_CT_Shuttle_to_BR.asStruct[mv_i].bCommand.dirFarward := TRUE;
            gMoverAxis.Q_CT_Shuttle_to_BR.asStruct[mv_i].bCommand.dirReverse := FALSE;
        END_FOR

        step := 11;
    END_IF

11: // init all mover until they the first shuttle is found
    gMoverAxis.Q_CT_Track_to_BR.asStruct.bCommand.startMoverNumberingSequence := (HMI.enState <> enState.StateMANU);

    IF gMoverAxis.I_CT_Track_from_BR.asStruct.bStatus.allIdSet THEN
        gMoverAxis.Q_CT_Track_to_BR.asStruct.bCommand.setShuttleNumber      := FALSE;
        gMoverAxis.Q_CT_Track_to_BR.asStruct.bCommand.releaseUnknownShuttle := FALSE;
        step                                                                := 13;
    END_IF

    IF gMoverAxis.I_CT_Track_from_BR.asStruct.bStatus.unknownMoverAtTarget1 THEN
        IF TRUE (* first shuttle sensor *) OR (TRACK_SIMULATION AND CONST.USE_SIMULATION) THEN
            step := 12;
        ELSE
            gMoverAxis.Q_CT_Track_to_BR.asStruct.bCommand.releaseUnknownShuttle := TRUE;
        END_IF
    ELSE
        gMoverAxis.Q_CT_Track_to_BR.asStruct.bCommand.releaseUnknownShuttle := FALSE;
    END_IF

12: // set all id since the first is found
    IF gMoverAxis.I_CT_Track_from_BR.asStruct.bStatus.unknownMoverAtTarget1 THEN
        gMoverAxis.Q_CT_Track_to_BR.asStruct.bCommand.setShuttleNumber := TRUE;
    ELSE
        gMoverAxis.Q_CT_Track_to_BR.asStruct.bCommand.setShuttleNumber := FALSE;
    END_IF

    IF gMoverAxis.I_CT_Track_from_BR.asStruct.bStatus.allIdSet THEN
        gMoverAxis.Q_CT_Track_to_BR.asStruct.bCommand.setShuttleNumber      := FALSE;
        gMoverAxis.Q_CT_Track_to_BR.asStruct.bCommand.releaseUnknownShuttle := FALSE;
        step                                                                := 13;
    END_IF

13: // stop id attrib sequence
    gMoverAxis.Q_CT_Track_to_BR.asStruct.bCommand.startMoverNumberingSequence := FALSE;
    step                                                                      := 14;

14: // check parameter
    // TODO here we have clearly somthing that will not work
    // when using groups... Groups should use the first station to set the waiting position
    // of the whole group
    IF THIS^.CheckWaitPosNotBehindStation() THEN
        ASSERT(0);
    END_IF

    gMoverAxis.Q_CT_Track_to_BR.asStruct.bCommand.enableProcess := TRUE;
    step                                                        := 15;

15: //move every shuttle to the last station
    FOR mv_i := 1 TO CONST.MOVER_NUMBER BY 1 DO
        _MoverList[mv_i].SetStation(THIS^._StationList[1]);
        _MoverList[mv_i].MoveToStation();

        _MoverList[mv_i].GetPiece(PiecePos_e.Assembly_left).UnloadPiece();
        _MoverList[mv_i].GetPiece(PiecePos_e.Assembly_right).UnloadPiece();
        _MoverList[mv_i].GetPiece(PiecePos_e.Test_left).UnloadPiece();
        _MoverList[mv_i].GetPiece(PiecePos_e.Test_right).UnloadPiece();

        _MoverList[mv_i].GetPiece(PiecePos_e.Assembly_left).Load();
        _MoverList[mv_i].GetPiece(PiecePos_e.Assembly_right).Load();
        _MoverList[mv_i].GetPiece(PiecePos_e.Test_left).Load();
        _MoverList[mv_i].GetPiece(PiecePos_e.Test_right).Load();
    END_FOR

    THIS^._WorkStationList.ApplyNewPath(ADR(THIS^._StationList),
                                        ADR(PERS.arrStationUsedList[PERS.iRecipeCurrent]),
                                        THIS^._PieceHolderList[1]);

    step := 16;

16:
    IF HMI_send_all_shuttle_to_unload THEN
        step := 15;
    END_IF
// do nothing, init done

END_CASE

(* ---------------------------------------------------------------------------- *)

// should be done elsewhere ...
SIMU.lrAccelMover := SIMU.lrAccelMoverSlider * SIMU.lrAccelMoverSlider;

RT_apply_station_list(CLK :=); // set by the HMI

IF RT_apply_station_list.Q OR (old_recipe <> PERS.iRecipeCurrent) THEN
    THIS^._WorkStationList.ApplyNewPath(ADR(THIS^._StationList),
                                        ADR(PERS.arrStationUsedList[PERS.iRecipeCurrent]),
                                        THIS^._PieceHolderList[1]);

    old_recipe := PERS.iRecipeCurrent;
END_IF

//Affect station offset depending on the station offset list
FOR mv_i := 1 TO CONST.STATION_NUMBER BY 1 DO
    _StationList[mv_i].Offset := PERS.arrStationOffsetsList[PERS.iRecipeCurrent][mv_i];
END_FOR

FOR mv_i := 1 TO CONST.MOVER_NUMBER BY 1 DO
    IF HMI.enState = enState.StateAUTO OR HMI.enState = enState.StateSTEP OR HMI.enState = enState.StateLEER THEN

        CASE _MoverList[mv_i].State OF

        MoverState_e.OperationDone:
            IF __ISVALIDREF(_MoverList[mv_i].Station.Process) THEN
                _MoverList[mv_i].Station.Process.TakeMover();
            ELSE
                ASSERT(0);
            END_IF

            _MoverList[mv_i].SetStation(_WorkStationList.GetNextStation(_MoverList[mv_i].Station));

        MoverState_e.WaitOnNextStation:
            // depending on the next station scenario, move
            CASE _MoverList[mv_i].Station.ApproachScenario OF
            // do not wait
            ApproachScenario_e.DoNotWait:
                _MoverList[mv_i].MoveToStation();

            // wait on the next station to be free
            ApproachScenario_e.WaitOnFinishedProcess:
                // Are we in a waiting spot ?
                IF __ISVALIDREF(_MoverList[mv_i].Station.Process) THEN

                    iNumOfMoverOnTheWay := THIS^.GetNumOfMoverOnTheWay(_MoverList[mv_i]);

                    IF 0 = iNumOfMoverOnTheWay THEN
                        _MoverList[mv_i].MoveToStation();

                    ELSIF iNumOfMoverOnTheWay <= _MoverList[mv_i].Station.iMaxWaitingMovers THEN
                        _MoverList[mv_i].MoveToWaitSpot();
                    END_IF

                ELSE
                    _MoverList[mv_i]
                        .SetStation(_WorkStationList.GetNextStationWithProcess(_MoverList[mv_i].Station));
                END_IF

            ApproachScenario_e.WaitOnFreeStation:

                IF NOT THIS^.IsMoverInRange(_MoverList[mv_i].MoverAxis.CurrentPos + (CONST.MAX_MOVER_SIZE / 2.0),
                                            _MoverList[mv_i].Station.Position.lrWorkPosition + CONST.MAX_MOVER_SIZE)
                    THEN
                    _MoverList[mv_i].MoveToStation();

                END_IF

            // wait on the previous station to be free (syncronize with the previous)
            ApproachScenario_e.WaitOnPrevProcess:
                // TODO implement !!!!
                _MoverList[mv_i].MoveToStation();

            // Move the mover only when all movers process are finished
            ApproachScenario_e.WaitOnExternalTrigger:
                IF bMoverSync THEN
                    // move only when there are no mover currently going to the station
                    IF NOT THIS^.IsMoverMovingToStation(mv_i) THEN
                        _MoverList[mv_i].MoveToStation();
                    END_IF
                END_IF

            END_CASE

        MoverState_e.WaitLeaveCurrentStation:
            IF NOT CONST.BIND_WITH_TRACK THEN
                _MoverList[mv_i].State := MoverState_e.MovingToStation;
            ELSE
                IF NOT gMoverAxis.I_CT_Shuttle_from_BR.asStruct[mv_i].bStatus.at_target THEN
                    _MoverList[mv_i].State := MoverState_e.MovingToStation;
                    // TODO need a fix to prevent a mover to be stucked here
                END_IF
            END_IF

        MoverState_e.MovingToStation:
            IF _MoverList[mv_i].IsInStationPos() THEN
                _MoverList[mv_i].State := MoverState_e.InStationPos;

            ELSIF NOT __ISVALIDREF(_MoverList[mv_i].Station) THEN
                ASSERT(0);
                _MoverList[mv_i].State := MoverState_e.WaitOnNextStation;
                _MoverList[mv_i].SetStation(_WorkStationList.GetNextStation(_MoverList[mv_i].Station));

            ELSIF __ISVALIDREF(_MoverList[mv_i].Station.Process) AND NOT CONST.BIND_WITH_TRACK THEN
                iNumOfMoverOnTheWay := THIS^.GetNumOfMoverOnTheWay(_MoverList[mv_i]);

                IF _MoverList[mv_i].Station.Process.xMoverPathFree AND
                   NOT (_MoverList[mv_i].Station.Equals(THIS^.GetNextMover(_MoverList[mv_i]).Station)) AND
                   (iNumOfMoverOnTheWay <= _MoverList[mv_i].Station.iMaxWaitingMovers) THEN
                    _MoverList[mv_i].MoveToStation();
                END_IF

            ELSIF _MoverList[mv_i].MoverAxis.isInPos AND NOT CONST.BIND_WITH_TRACK THEN
                _MoverList[mv_i].MoveToStation();
            END_IF

        MoverState_e.InStationPos:
            IF NOT __ISVALIDREF(_MoverList[mv_i].Station) THEN
                ASSERT(0);
                _MoverList[mv_i].State := MoverState_e.WaitOnNextStation;
                _MoverList[mv_i].SetStation(_WorkStationList.GetNextStation(_MoverList[mv_i].Station));

                // If there is no station (waiting position)
            ELSIF NOT __ISVALIDREF(_MoverList[mv_i].Station.Process) THEN
                _MoverList[mv_i].State := MoverState_e.WaitOnNextStation;
                _MoverList[mv_i].SetStation(_WorkStationList.GetNextStation(_MoverList[mv_i].Station));

            ELSE
                IF __ISVALIDREF(_MoverList[mv_i].Station.Process.Mover) THEN
                    // ASSERT(0); TODO we have to find why we are here so often.

                    IF _MoverList[mv_i].Station.Process.xMoverShouldLeave THEN
                        _MoverList[mv_i].Station.Process.TakeMover();
                        ASSERT(0);

                    ELSE
                        _MoverList[mv_i].State := MoverState_e.OperationDone;
                    END_IF
                ELSE
                    _MoverList[mv_i].Station.Process.GiveMover(_MoverList[mv_i]);
                    _MoverList[mv_i].State := MoverState_e.InOperation;
                END_IF
            END_IF

        MoverState_e.InOperation:
            IF NOT __ISVALIDREF(_MoverList[mv_i].Station) THEN
                ASSERT(0);
                _MoverList[mv_i].State := MoverState_e.WaitOnNextStation;
                _MoverList[mv_i].SetStation(_WorkStationList.GetNextStation(_MoverList[mv_i].Station));

            ELSIF NOT __ISVALIDREF(_MoverList[mv_i].Station.Process) THEN
                ASSERT(0);
                _MoverList[mv_i].State := MoverState_e.OperationDone;

            ELSIF _MoverList[mv_i].Station.Process.xMoverShouldLeave THEN
                _MoverList[mv_i].State := MoverState_e.OperationDone;

            ELSIF NOT __ISVALIDREF(_MoverList[mv_i].Station.Process.Mover) THEN
                ASSERT(0);
                _MoverList[mv_i].Station.Process.GiveMover(_MoverList[mv_i]);

            ELSIF (__ISVALIDREF(_MoverList[mv_i].Station.Process.Mover) AND_THEN
                   (_MoverList[mv_i].Station.Process.Mover._id <> mv_i)) THEN
                ASSERT(0);
                _MoverList[mv_i].Station.Process.Mover.Abort(_StationList[1]);
                _MoverList[mv_i].Station.Process.GiveMover(_MoverList[mv_i]);
            END_IF

        MoverState_e.PerformRelativeMove:
            IF NOT __ISVALIDREF(_MoverList[mv_i].Station) THEN
                ASSERT(0);
                _MoverList[mv_i].State := MoverState_e.WaitOnNextStation;
                _MoverList[mv_i].SetStation(_WorkStationList.GetNextStation(_MoverList[mv_i].Station));

            ELSIF NOT __ISVALIDREF(_MoverList[mv_i].Station.Process) THEN
                ASSERT(0);
                _MoverList[mv_i].State := MoverState_e.OperationDone;

            ELSIF _MoverList[mv_i].Station.Process.xMoverShouldLeave THEN
                _MoverList[mv_i].State := MoverState_e.OperationDone;

            ELSE
                IF NOT _MoverList[mv_i].IsInStationPos() THEN
                    _MoverList[mv_i].State := MoverState_e.WaitRelativeMoveEnd;
                END_IF

            END_IF

        MoverState_e.WaitRelativeMoveEnd:
            IF NOT __ISVALIDREF(_MoverList[mv_i].Station) THEN
                ASSERT(0);
                _MoverList[mv_i].State := MoverState_e.WaitOnNextStation;
                _MoverList[mv_i].SetStation(_WorkStationList.GetNextStation(_MoverList[mv_i].Station));

            ELSIF NOT __ISVALIDREF(_MoverList[mv_i].Station.Process) THEN
                ASSERT(0);
                _MoverList[mv_i].State := MoverState_e.OperationDone;

            ELSE
                IF _MoverList[mv_i].IsInStationPos() THEN
                    _MoverList[mv_i].State := MoverState_e.InOperation;

                ELSIF gMoverAxis.I_CT_Shuttle_from_BR.asStruct[mv_i].bStatus.at_target THEN
                    _MoverList[mv_i].State := MoverState_e.PerformRelativeMove;
                END_IF

            END_IF

        END_CASE
    END_IF
END_FOR

// update bMoverSync
bMoverSync := THIS^.IsAllMoverAtPosition() OR THIS^.IsMoverStucked();

// start update simu mover **********************************************
IF CONST.USE_SIMULATION THEN
    FOR mv_i := 1 TO CONST.MOVER_NUMBER BY 1 DO
        _MoverList[mv_i].MoverAxis(xIN_StopMover := HMI_xStopMover);
    END_FOR
END_IF

// stop update simu mover **********************************************

// start communication with B&R PLC ************************************
gMoverAxis.Q_CT_Track_to_BR.asStruct.bCommand.force_IDSet :=
    NOT gMoverAxis.I_CT_Track_from_BR.asStruct.bStatus.allIdSet AND
    ((11 = step) OR (12 = step) OR (13 = step)) AND
    THIS^.IsAllIDSet();

fb_Bp_Enable_Power(pbtIN := ADR(HMI_Bp_Enable_Power),
                   xINon := gMoverAxis.Q_CT_Track_to_BR.asStruct.bCommand.enablePower);

fb_Bp_Enable_Process(pbtIN := ADR(HMI_Bp_Enable_Process),
                     xINon := gMoverAxis.Q_CT_Track_to_BR.asStruct.bCommand.enableProcess);

// track control
IF CONST.BIND_WITH_TRACK THEN
    // Quit
    gMoverAxis.Q_CT_Track_to_BR.asStruct.bCommand.resetErrors := HMI.btArMain[7].press;

    IF ((enState.StateMANU = HMI.enState) AND HMI_Bp_Enable_Power.rtrig) THEN
        gMoverAxis.Q_CT_Track_to_BR.asStruct.bCommand.enablePower :=
            NOT gMoverAxis.Q_CT_Track_to_BR.asStruct.bCommand.enablePower;
    END_IF

    IF ((enState.StateMANU = HMI.enState) AND HMI_Bp_Enable_Process.rtrig) THEN
        gMoverAxis.Q_CT_Track_to_BR.asStruct.bCommand.enableProcess :=
            NOT gMoverAxis.Q_CT_Track_to_BR.asStruct.bCommand.enableProcess;
    END_IF

    // This should be a temporary fix to be sure that the ST120 axis is up before
    // any shuttle is allowed to run
    IF (_14_STATE.fb_State.xIN_InitEND) THEN
        gMoverAxis.Q_CT_Track_to_BR.asStruct.bCommand.enablePower := TRUE;
    ELSIF HMI.enState < enState.StateREADY AND (enState.StateMANU <> HMI.enState) THEN
        gMoverAxis.Q_CT_Track_to_BR.asStruct.bCommand.enablePower := FALSE;
    END_IF

ELSE
    gMoverAxis.I_CT_Track_from_BR.asStruct.bStatus.allIdSet := TRUE;

END_IF

// shuttle control
IF CONST.BIND_WITH_TRACK AND gMoverAxis.Q_CT_Track_to_BR.asStruct.bCommand.enableProcess THEN

    FOR mv_i := 1 TO CONST.MOVER_NUMBER BY 1 DO
        IF __ISVALIDREF(_MoverList[mv_i].Station) THEN
            gMoverAxis.Q_CT_Shuttle_to_BR.asStruct[mv_i].bCommand.release :=
                ((THIS^._MoverList[mv_i].State = MoverState_e.WaitLeaveCurrentStation) OR
                (_MoverList[mv_i].State = MoverState_e.MovingToStation) OR
                (_MoverList[mv_i].State = MoverState_e.PerformRelativeMove)) AND
                gMoverAxis.I_CT_Shuttle_from_BR.asStruct[mv_i].bStatus.at_target;

            gMoverAxis.Q_CT_Shuttle_to_BR.asStruct[mv_i].bNextStation    := _MoverList[mv_i].Station.SuperTrackNumber;
            gMoverAxis.Q_CT_Shuttle_to_BR.asStruct[mv_i].diNextOffset_um :=
                LREAL_TO_DINT(_MoverList[mv_i].Station.Offset * 1000.0 +
                              _MoverList[mv_i].MovingProcessOffset * 1000.0);

            // echo At_Target
            gMoverAxis.Q_CT_Shuttle_to_BR.asStruct[mv_i].bCommand.echo_At_Target :=
                gMoverAxis.I_CT_Shuttle_from_BR.asStruct[mv_i].bStatus.at_target;

            // echo at position
            gMoverAxis.Q_CT_Shuttle_to_BR.asStruct[mv_i].bCommand.echo_in_pos :=
                gMoverAxis.I_CT_Shuttle_from_BR.asStruct[mv_i].bStatus.in_position;

        END_IF
    END_FOR
END_IF

// stop communication with B&R PLC ************************************

// test if path is free
IF CONST.BIND_WITH_TRACK THEN
    gMoverAxis.Q_CT_Track_to_BR.asStruct.bCommand.wholePathFree := TRUE;

    FOR mv_i := 1 TO CONST.STATION_NUMBER BY 1 DO
        IF __ISVALIDREF(_StationList[mv_i].Process) AND_THEN NOT _StationList[mv_i].Process.xMoverPathFree THEN
            gMoverAxis.Q_CT_Track_to_BR.asStruct.bCommand.wholePathFree := FALSE;
        END_IF
    END_FOR

    IF HMI.enState = enState.StateMANU THEN
        gMoverAxis.Q_CT_Track_to_BR.asStruct.bCommand.wholePathFree := TRUE;
    END_IF
END_IF

// start collision check **********************************************
IF NOT CONST.BIND_WITH_TRACK THEN
    FOR mv_i := 1 TO CONST.MOVER_NUMBER - 1 BY 1 DO
        _MoverList[mv_i].MoverAxis.IsColliding(_MoverList[mv_i + 1].MoverAxis);
        _MoverList[mv_i].MoverAxis.WillCollide(_MoverList[mv_i + 1].MoverAxis);

        IF THIS^.IsMoverLost(THIS^._MoverList[mv_i]) THEN
            // ASSERT HERE, WE SHOULD NEVER GO HERE
            // ASSERT(0);
        END_IF
    END_FOR

    _MoverList[CONST.MOVER_NUMBER].MoverAxis
        .IsColliding(_MoverList[1].MoverAxis); // do not forget to test this case, too

    _MoverList[CONST.MOVER_NUMBER].MoverAxis.WillCollide(_MoverList[1].MoverAxis);
END_IF

// end collision check **********************************************

// start output affectation **********************************************
xOUT_AllMoverEmpty := TRUE;

FOR mv_i := 1 TO CONST.MOVER_NUMBER BY 1 DO
    // IF (F_GetHighestStationDoneAssembly(_MoverList[mv_i]) <> 0) OR
    //    (F_GetHighestStationDoneTest(_MoverList[mv_i]) <> 0) THEN
    IF FALSE THEN
        xOUT_AllMoverEmpty := FALSE;
    END_IF
END_FOR

xOUT_Error := gMoverAxis.I_CT_Track_from_BR.asStruct.bStatus.error AND CONST.BIND_WITH_TRACK;

// end output affectation **********************************************

// This method check if the wait pos of a given station is before another
// station. This situation is not permitted by the system, yet
METHOD CheckWaitPosNotBehindStation : BOOL
VAR_INPUT
END_VAR
VAR
    i : INT;
END_VAR
CheckWaitPosNotBehindStation := FALSE;
FOR i := 2 TO CONST.STATION_NUMBER BY 1 DO
    CheckWaitPosNotBehindStation := CheckWaitPosNotBehindStation OR
        THIS^._StationList[i].Position.lrWorkPosition + THIS^._StationList[i].WaitPos <
        THIS^._StationList[i - 1].Position.lrWorkPosition;
END_FOR

// NO CHECK ARE MADE BETWEEN THE FIRST POS AND THE LAST
END_METHOD

METHOD Equals : BOOL
VAR_INPUT
    object : ANY;
END_VAR
Equals := THIS = object.pValue;
END_METHOD

METHOD FB_init : BOOL
VAR_INPUT
    bInitRetains : BOOL; // if TRUE, the retain variables are initialized (warm start / cold start)
    bInCopyCode  : BOOL; // if TRUE, the instance afterwards gets moved into the copy code (online change)
END_VAR
VAR
    i : INT;
END_VAR
THIS^._iID := THIS^._iInstanceCounter;
THIS^._iInstanceCounter := THIS^._iInstanceCounter +1;
END_METHOD

METHOD PUBLIC GetAllMoverPos : BOOL
VAR_INPUT
    my_mover_list : REFERENCE TO ARRAY[1..CONST.MOVER_NUMBER] OF MoverDict;
END_VAR
VAR
    index : INT;
END_VAR
FOR index := 1 TO CONST.MOVER_NUMBER BY 1 DO
    my_mover_list[index].MoverNum := index;
    my_mover_list[index].MoverPos := THIS^._MoverList[index].MoverAxis.CurrentPos;
END_FOR
END_METHOD

METHOD PUBLIC GetAllStationPos : BOOL
VAR_INPUT
    my_mover_list : REFERENCE TO ARRAY[1..CONST.STATION_NUMBER] OF StationDict;
END_VAR
VAR
    index : INT;
END_VAR
FOR index := 1 TO CONST.STATION_NUMBER BY 1 DO
    my_mover_list[index].StationNum := index;
    my_mover_list[index].StationPos := THIS^._StationList[index].Position.lrWorkPosition;
END_FOR
END_METHOD

METHOD GetMoverIndex : INT
VAR_INPUT
    mover : REFERENCE TO FB_Mover;
END_VAR
VAR
    i : INT;
END_VAR
FOR i:= 1 TO CONST.MOVER_NUMBER BY 1 DO 
	IF mover.Equals(THIS^._MoverList[i]) THEN
		GetMoverIndex := i;
		EXIT;
	END_IF
END_FOR
END_METHOD

// Is a shuttle present in the given region?
// If 'from_pos' is greater than 'to_pos', this means we look in
// a region that include the begining of the track
METHOD PUBLIC GetMoverInRange : REFERENCE TO FB_Mover
VAR_INPUT
    from_pos : LREAL; // begin of the tested region (included)
    to_pos   : LREAL; // end of the tested region (included)
END_VAR
VAR
    i : INT;
END_VAR

GetMoverInRange REF= 0;

IF from_pos < to_pos THEN
    FOR i := 1 TO CONST.MOVER_NUMBER BY 1 DO
        IF (THIS^._MoverList[i].MoverAxis.CurrentPos >= from_pos) AND
           (THIS^._MoverList[i].MoverAxis.CurrentPos <= to_pos) THEN
            GetMoverInRange REF= THIS^._MoverList[i];
            EXIT;

        END_IF
    END_FOR
ELSE // we test a region that pass by the maximum track length
    FOR i := 1 TO CONST.MOVER_NUMBER BY 1 DO
        IF (THIS^._MoverList[i].MoverAxis.CurrentPos >= from_pos) OR
           (THIS^._MoverList[i].MoverAxis.CurrentPos <= to_pos) THEN
            GetMoverInRange REF= THIS^._MoverList[i];
            EXIT;

        END_IF
    END_FOR
END_IF
END_METHOD

// Get the position of a given mover using its index number
METHOD PUBLIC GetMoverPosFromIndex : LREAL
VAR_INPUT
    MoverIndex : INT;
END_VAR
IF (MoverIndex < 1) OR (MoverIndex > CONST.MOVER_NUMBER) THEN
	GetMoverPosFromIndex := 0.0;
ELSE
	GetMoverPosFromIndex := THIS^._MoverList[MoverIndex].MoverAxis.CurrentPos;
END_IF
END_METHOD

// Get the mover with the next number (Means the mover behind)
METHOD GetNextMover : REFERENCE TO FB_Mover
VAR_INPUT
    Mover : REFERENCE TO FB_Mover;
END_VAR
VAR
    moverIndex : INT;
END_VAR
moverIndex := THIS^.GetMoverIndex(Mover);

IF moverIndex >= CONST.MOVER_NUMBER THEN
    GetNextMover REF= THIS^._MoverList[1];
ELSE
    GetNextMover REF= THIS^._MoverList[moverIndex + 1];
END_IF
END_METHOD

// we check if there is a mover between refMover and the refMover.Station
// This method is used to unblock a mover that cannot move because of a mover
// "Behind" it that also want to move to the same station
METHOD PRIVATE GetNumOfMoverOnTheWay : INT
VAR_INPUT
    refMover : REFERENCE TO FB_Mover; // The maybe stucking mover
END_VAR
VAR
    lrMoverPosTemp   : LREAL; // we use this position beacuse maybe we are at the end of the track
    lrStationPosTemp : LREAL; // we use this position beacuse maybe we are at the end of the track
    i                : INT;
END_VAR
GetNumOfMoverOnTheWay := 0;

FOR i := 1 TO CONST.MOVER_NUMBER BY 1 DO
    // If the mover is in front of the tested mover, we add MAX_TRACK_LENGTH (maybe we are at the end of the track ?)
    IF refMover.IsInFront(THIS^._MoverList[i].MoverAxis.CurrentPos) THEN
        lrMoverPosTemp := THIS^._MoverList[i].MoverAxis.CurrentPos + CONST.MAX_TRACK_LENGTH;
    ELSE
        lrMoverPosTemp := THIS^._MoverList[i].MoverAxis.CurrentPos;
    END_IF

    // If the mover is in front of the station, we add MAX_TRACK_LENGTH (maybe we are at the end of the track ?)
    IF refMover.IsInFront(refMover.Station.Position.lrWorkPosition) THEN
        lrStationPosTemp := refMover.Station.Position.lrWorkPosition + CONST.MAX_TRACK_LENGTH;
    ELSE
        lrStationPosTemp := refMover.Station.Position.lrWorkPosition;
    END_IF

    IF (lrMoverPosTemp > refMover.MoverAxis.CurrentPos) AND
       (lrMoverPosTemp <= lrStationPosTemp) THEN
	   // If a mover is at position but has
        GetNumOfMoverOnTheWay := GetNumOfMoverOnTheWay + 1;
    END_IF
END_FOR
END_METHOD

// Get the mover with the previous number (Means the front mover)
METHOD GetPrevMover : REFERENCE TO FB_Mover
VAR_INPUT
    Mover : REFERENCE TO FB_Mover;
END_VAR
VAR
    moverIndex : INT;
END_VAR
moverIndex := THIS^.GetMoverIndex(Mover);

IF moverIndex <= 1 THEN
    GetPrevMover REF= THIS^._MoverList[CONST.MOVER_NUMBER];
ELSE
    GetPrevMover REF= THIS^._MoverList[moverIndex - 1];
END_IF

IF GetPrevMover.MoverAxis.CurrentPos < Mover.MoverAxis.CurrentPos THEN
	GetPrevMover REF= THIS^.GetNextMover(Mover);
END_IF
END_METHOD

METHOD PRIVATE IsAllIDSet : BOOL
VAR_INPUT
END_VAR
VAR
    i : INT;
    j : INT;
END_VAR
IsAllIDSet := TRUE;

FOR i := 1 TO CONST.MOVER_NUMBER - 1 BY 1 DO

    FOR j := i + 1 TO CONST.MOVER_NUMBER BY 1 DO
        IsAllIDSet := IsAllIDSet AND
                      (THIS^._MoverList[i].MoverAxis.CurrentPos <> THIS^._MoverList[j].MoverAxis.CurrentPos);
    END_FOR

END_FOR
END_METHOD

METHOD IsAllMoverAtPosition : BOOL
VAR_INPUT
END_VAR
VAR
    i : INT;
END_VAR
IsAllMoverAtPosition := TRUE;

FOR i := 1 TO CONST.MOVER_NUMBER BY 1 DO
    IF (THIS^._MoverList[i].State = MoverState_e.WaitLeaveCurrentStation) OR
       (THIS^._MoverList[i].State = MoverState_e.MovingToStation) OR
       (THIS^._MoverList[i].State = MoverState_e.InStationPos) THEN
        IsAllMoverAtPosition := FALSE;
        EXIT;
    END_IF
END_FOR
END_METHOD

// Is a shuttle present in the given region?
// If 'from_pos' is greater than 'to_pos', this means we look in
// a region that include the begining of the track
METHOD PUBLIC IsMoverInRange : BOOL
VAR_INPUT
    from_pos : LREAL; // begin of the tested region (included)
    to_pos   : LREAL; // end of the tested region (included)
END_VAR
VAR
    i : INT;
END_VAR
IsMoverInRange := __ISVALIDREF(THIS^.GetMoverInRange(from_pos, to_pos));
END_METHOD

// If the target station of a mover is not between the target of the previous and the next mover
// this function will return true. This function is attendend to debug only
METHOD IsMoverLost : BOOL
VAR_INPUT
    mover : REFERENCE TO FB_Mover;
END_VAR
VAR
    i : INT;

    prevStationLoc  : LREAL;
    nextStationLoc  : LREAL;
    moverStationLoc : LREAL; // mover to test location
    posList         : ARRAY[0..2] OF LREAL;
END_VAR
(* the algorithm function as fallow 

First we built a sorted array based on the station position
Then we search for the previous station position and fix
our search index
Then we check if the squence of mover is correct. The sequence must be
PreviousMoverStation -> CurrentMoverStation -> NextMoverStation
If we don't get this sequence, then the mover is lost.

In fact, since we have only 3 elements, we only need to check
the next station
*)
IsMoverLost := FALSE;

nextStationLoc  := THIS^.GetNextMover(mover).Station.Position.lrWorkPosition;
prevStationLoc  := THIS^.GetPrevMover(mover).Station.Position.lrWorkPosition;
moverStationLoc := mover.station.Position.lrWorkPosition;

posList[0] := prevStationLoc;
posList[1] := moverStationLoc;
posList[2] := nextStationLoc;

SortBubbleLREAL(ADR(posList), 0, 2);

IF posList[0] = prevStationLoc THEN
    IF posList[1] <> moverStationLoc THEN
        IsMoverLost := TRUE;
    END_IF

ELSIF posList[0] = moverStationLoc THEN
    IF posList[1] <> nextStationLoc THEN
        IsMoverLost := TRUE;
    END_IF

ELSE (* posList[0] = nextStationLoc *)
    IF posList[1] <> prevStationLoc THEN
        IsMoverLost := TRUE;
    END_IF
END_IF
END_METHOD

METHOD PRIVATE IsMoverMovingToStation : BOOL
VAR_INPUT
    iMoverNumber : INT; // the current mover number 
END_VAR
VAR
    i           : INT;
END_VAR
IsMoverMovingToStation := FALSE;

FOR i := 1 TO CONST.MOVER_NUMBER BY 1 DO

    // we don't check the tests mover station, else it will be always true
    IF (iMoverNumber <> i) AND THIS^._MoverList[i].Station.Equals(THIS^._MoverList[iMoverNumber].Station) THEN
        IsMoverMovingToStation := IsMoverMovingToStation OR
                                  (THIS^._MoverList[i].State = MoverState_e.WaitLeaveCurrentStation) OR
                                  (THIS^._MoverList[i].State = MoverState_e.MovingToStation) OR
                                  (THIS^._MoverList[i].State = MoverState_e.InStationPos);

        // Do not exit here, since we OR the flag
        // TODO maybe we should add an IF statement to exit when the flag is true
        // because it will never be false again ... ? // PERFORMANCE ISSUE
    END_IF

END_FOR
END_METHOD

// Return TRUE if at least one mover is stucked
METHOD IsMoverStucked : BOOL
VAR_INPUT
END_VAR
IsMoverStucked := FALSE;

FOR mv_i := 1 TO CONST.MOVER_NUMBER BY 1 DO
    IF THIS^._MoverList[mv_i].MoverAxis.xStuck THEN
        IsMoverStucked := TRUE;
        EXIT;
    END_IF
END_FOR
END_METHOD

// Is the given process used by the current station configuration?
METHOD IsProcessUsed : BOOL
VAR_INPUT
    this_process : REFERENCE TO FB_AUT_ABSTRACT;
END_VAR
VAR
	i : INT;
END_VAR
IsProcessUsed := THIS^._WorkStationList.IsProcessUsed(this_process);
END_METHOD

METHOD SetAllScenario : REFERENCE TO FB_MoverMan
VAR_INPUT
END_VAR
VAR
	i : INT;
END_VAR
FOR i := 1 TO CONST.STATION_NUMBER BY 1 DO
    THIS^._StationList[i].ApproachScenario := THIS^.HMI_Scenario;
END_FOR

SetAllScenario REF= THIS^;
END_METHOD

// Give a random time for each process. It ensure at least the minimum and the maximum value are given
// to at least 2 diffrents process
METHOD SetAllTimers : REFERENCE TO FB_MoverMan
VAR_INPUT
    arrStationTime : POINTER TO DINT;
    udiOffset      : UDINT; // simple offset to apply to the seed
END_VAR
VAR
    i         : INT;
    rand      : DRAND;
    tempIndex : INT := 0;
    getTime   : GETSYSTEMTIME;
END_VAR
IF arrStationTime <> 0 THEN
	
    getTime();
    rand.Seed := TO_INT(getTime.timeLoDW + udiOffset);

    FOR i := 0 TO CONST.STATION_NUMBER - 1 BY 1 DO
        rand();
        arrStationTime[i] := TO_DINT((THIS^.HMI_TimeMax - THIS^.HMI_TimeMin) * (rand.Num) + THIS^.HMI_TimeMin);
    END_FOR

    tempIndex := 0;

    FOR i := 1 TO CONST.STATION_NUMBER - 1 BY 1 DO
        IF arrStationTime[i] < arrStationTime[tempIndex] THEN
            tempIndex := i;
        END_IF
    END_FOR

    arrStationTime[tempIndex] := THIS^.HMI_TimeMin;

    tempIndex := 0;

    FOR i := 1 TO CONST.STATION_NUMBER - 1 BY 1 DO
        IF arrStationTime[i] > arrStationTime[tempIndex] THEN
            tempIndex := i;
        END_IF
    END_FOR

    arrStationTime[tempIndex] := THIS^.HMI_TimeMax;
END_IF

SetAllTimers REF= THIS^;
END_METHOD

METHOD ToString : STRING
VAR_INPUT
END_VAR
ToString := CONCAT('FB_MoverMan_', TO_STRING(THIS^._iID));
END_METHOD

END_FUNCTION_BLOCK

// ---- POUs/20_AUTO/Mover/FB_PieceHolderMover.TcPOU
FUNCTION_BLOCK FB_PieceHolderMover EXTENDS FB_BasePieceHolder IMPLEMENTS IObject
VAR_INPUT
END_VAR
VAR_OUTPUT
END_VAR
VAR
	_lrPosOffset : LREAL; // current offset position
    _Piece       : FB_My_Piece;
	
	_iID : INT := 0; // instance ID, is set during FB_Init using the value of _iInstanceCounter 
END_VAR
VAR_STAT
	_iInstanceCounter : INT := 1; // instance counter
END_VAR

METHOD Equals : BOOL
VAR_INPUT
    object : ANY;
END_VAR
Equals := THIS = object.pValue;
END_METHOD

METHOD FB_init : BOOL
VAR_INPUT
    bInitRetains : BOOL;  // if TRUE, the retain variables are initialized (warm start / cold start)
    bInCopyCode  : BOOL;  // if TRUE, the instance afterwards gets moved into the copy code (online change)
    offset       : LREAL; //position offset of the tool using this toolhead, a negative value represents a move on the left
END_VAR
THIS^._iID := THIS^._iInstanceCounter;
THIS^._iInstanceCounter := THIS^._iInstanceCounter +1;
THIS^.PosOffset := 0;
END_METHOD

METHOD PUBLIC  GetPiece : REFERENCE TO FB_My_Piece
VAR_INPUT
END_VAR
GetPiece REF= THIS^._Piece;
END_METHOD

PROPERTY PosOffset : LREAL
GET
PosOffset := _lrPosOffset;
END_GET
SET
_lrPosOffset := PosOffset;
END_SET
END_PROPERTY

METHOD ToString : STRING
VAR_INPUT
END_VAR
ToString := CONCAT('FB_PieceHolder_', TO_STRING(THIS^._iID));
END_METHOD

END_FUNCTION_BLOCK

// ---- POUs/20_AUTO/Mover/FB_BasePieceHolder.TcPOU
FUNCTION_BLOCK FB_BasePieceHolder
VAR
    _Usable : BOOL := TRUE;
END_VAR

METHOD Equals : BOOL
VAR_INPUT
    object : ANY;
END_VAR
Equals := THIS = object.pValue;
END_METHOD

PROPERTY PUBLIC Usable : BOOL
GET
Usable := THIS^._Usable;
END_GET
SET
THIS^._Usable := Usable;
END_SET
END_PROPERTY

END_FUNCTION_BLOCK

// ---- POUs/20_AUTO/Mover/FB_My_Piece.TcPOU
// Piece description used in this project
FUNCTION_BLOCK PUBLIC FB_My_Piece EXTENDS FB_Piece
VAR_INPUT
END_VAR
VAR_OUTPUT
END_VAR
VAR
    // add special piece information here
END_VAR

METHOD PUBLIC UnloadPiece : BOOL
VAR_INPUT
END_VAR
SUPER^.UnloadPiece();
END_METHOD

END_FUNCTION_BLOCK

// ---- POUs/20_AUTO/Mover/FB_Piece.TcPOU
(* Abstract piece, need to be implemented 
 * for you project needs *)
FUNCTION_BLOCK PUBLIC FB_Piece
VAR
    _Exist           : BOOL := FALSE;
    _State           : PieceState_e;
    _LastStationDone : INT    := 0;
    _ErrorMessage    : STRING := '';

    _MarkMessage : STRING := ''; // use to know what is the message engraved in the piece
END_VAR

METHOD Equals : BOOL
VAR_INPUT
    object : ANY;
END_VAR
Equals := THIS = object.pValue;
END_METHOD

PROPERTY PUBLIC Exist : BOOL
GET
Exist := THIS^._Exist;
END_GET
END_PROPERTY

METHOD PUBLIC GetErrorMessage : STRING
VAR_INPUT
END_VAR
IF THIS^._Exist THEN
	GetErrorMessage := THIS^._ErrorMessage;
END_IF
END_METHOD

// Return the last station done
// The number returned is always positive
// Use IsBad() to know if a piece is bad
METHOD PUBLIC GetLastStationDone : INT
VAR_INPUT
END_VAR
IF THIS^._Exist THEN
    GetLastStationDone := ABS(THIS^._LastStationDone);
END_IF
END_METHOD

METHOD PUBLIC IsBad : BOOL
VAR_INPUT
END_VAR
IF THIS^._Exist THEN
    IsBad := (THIS^._LastStationDone < 0) OR (LEN(THIS^._ErrorMessage) > 0) OR (PieceState_e.bad = THIS^._State);
END_IF
END_METHOD

METHOD PUBLIC IsPieceInWorkingState : BOOL
VAR_INPUT
END_VAR
IsPieceInWorkingState := FALSE;

IF THIS^._Exist THEN
    IsPieceInWorkingState := PieceState_e.working = THIS^._State;
END_IF
END_METHOD

// Load a piece inside the pieceholder. The flag _Exists is set
METHOD PUBLIC Load : BOOL
VAR_INPUT
END_VAR
THIS^._Exist := TRUE;
END_METHOD

METHOD PUBLIC Mark : BOOL
VAR_INPUT
    Message : STRING;
END_VAR
IF THIS^._Exist THEN
    THIS^._MarkMessage := Message;
END_IF
END_METHOD

METHOD PUBLIC SetErrorMessage : BOOL
VAR_INPUT
	ErrorMessage : STRING;
END_VAR
IF LEN(THIS^._ErrorMessage) > 0 THEN
    SetErrorMessage := FALSE;
ELSE
	THIS^._ErrorMessage := ErrorMessage;
    THIS^.SetLastStation(- THIS^._LastStationDone);
END_IF
END_METHOD

/// Set the last station done
/// Call this method only once during the your process
/// This method will automatically update the piece state
/// from the Working state to the good or bad state depending of the error state
METHOD PUBLIC SetLastStation : BOOL
VAR_INPUT
    value : INT;
END_VAR
IF THIS^._Exist THEN
    IF ABS(value) < ABS(THIS^._LastStationDone) THEN
        SetLastStation := FALSE;
    ELSE
        IF THIS^._LastStationDone < 0 THEN
            value := 0 - ABS(value);
        END_IF

        THIS^._LastStationDone := value;

        IF THIS^._LastStationDone >= 0 THEN
            THIS^._State := PieceState_e.good;
        ELSE
            THIS^._State := PieceState_e.bad;
        END_IF

        SetLastStation := TRUE;
    END_IF
ELSE
    SetLastStation := FALSE;
END_IF
END_METHOD

METHOD PUBLIC StartWorking : BOOL
VAR_INPUT
END_VAR
IF PieceState_e.good = THIS^._State THEN
    THIS^._State := PieceState_e.working;
END_IF
END_METHOD

METHOD PUBLIC UnloadPiece : BOOL
VAR_INPUT
END_VAR
_Exist           := FALSE;
_State           := PieceState_e.good;
_LastStationDone := 0;
_ErrorMessage    := '';
_MarkMessage     := '';
END_METHOD

END_FUNCTION_BLOCK

// ---- POUs/20_AUTO/Mover/FB_SimuMoverAxis.TcPOU
FUNCTION_BLOCK FB_SimuMoverAxis IMPLEMENTS IObject
VAR_INPUT
    xIN_StopMover : BOOL; // stop the mover from movinf
END_VAR
VAR_OUTPUT
    outSimuCurrentPos   : Pos2D_t; // Mover position, expressed as slot number
    outSimuCurrentPosSC : Pos2D_t; // Mover position, expressed as pixel for SC
    outSimuCurrentRot   : INT;     // mover current rotation
    isInPos             : BOOL;    // true when targetPos = currentPos
END_VAR
VAR
    // with tick rate at 10ms, a value of 10 gives us 1m/s
    _Velocity    : LREAL := 0;     // Mover velocity, expressed as mm per tick, max is 10m/s
    _ErrorState  : INT   := 0;     // error state, not used
    _TargetPos   : LREAL := 0;     // last target pos
    _CurrentPos  : LREAL := 0;     // Current Pos, but with more resolution than the pixel
    _IsColliding : BOOL  := FALSE; // When true, the mover should not move
    _LastPos     : LREAL := 0;     // last position, used to trigger the xStuck flag
    _xStuck      : BOOL;           // true when the axis does not move
    _willCollide : BOOL := FALSE;  // TRUE if a collision will occure with the current velocity

    {attribute 'hide'}
    _lrNextStopPos : LREAL; // local variable used to get next stop

    _iID : INT := 0; // instance ID, is set during FB_Init using the value of _iInstanceCounter 

    _CurrentDir : MoverDirection_e := MoverDirection_e.Farward;
END_VAR

VAR_TEMP
    _MoverAccel : LREAL; // Mover acceleration, can be positive or negative depending on the direction
END_VAR

VAR CONSTANT
    MAX_POS  : LREAL := CONST.MAX_TRACK_LENGTH; // should be defined elsewhere ...
    MAX_SIZE : LREAL := CONST.MAX_MOVER_SIZE;   // Maxium size of the mover
    //MOVER_ACCEL        : LREAL := 0.1;                      // Mover acceleration, in mm/tick^2
    //MOVER_VELOCITY_MAX : LREAL := 20;                     // Mover velocity, expressed as mm per tick, max is 10m/s
    MOVER_VELOCITY_MIN : LREAL := 1.0; // Mover velocity, expressed as mm per tick, max is 10m/s
END_VAR
VAR_STAT
    _iInstanceCounter : INT := 1; // instance counter
END_VAR

IF NOT xIN_StopMover THEN // Do not change momemtum when we stop the movers from HMI
    IF MoverDirection_e.Farward = THIS^._CurrentDir THEN
        _MoverAccel := SIMU.lrAccelMover;
    ELSE
        _MoverAccel := -SIMU.lrAccelMover;
    END_IF

    IF NOT _IsColliding THEN

        IF THIS^.GetStopLen(_Velocity, SIMU.lrAccelMover) >= DistToTravel(_CurrentPos, _TargetPos) OR
           THIS^._willCollide THEN
            _Velocity := _Velocity - _MoverAccel;

        ELSIF SIMU.lrSpeedMover > ABS(_Velocity) AND _CurrentPos <> _TargetPos THEN
            _Velocity := _Velocity + _MoverAccel;

        END_IF
    ELSE
        _Velocity := _Velocity - _MoverAccel;
    END_IF
END_IF

// protect max and min speed
IF SIMU.lrSpeedMover < ABS(_Velocity) THEN
    IF MoverDirection_e.Farward = THIS^._CurrentDir THEN
        _Velocity := SIMU.lrSpeedMover;
    ELSE
        _Velocity := -SIMU.lrSpeedMover;
    END_IF
ELSIF ABS(_Velocity) < MOVER_VELOCITY_MIN THEN
    IF MoverDirection_e.Farward = THIS^._CurrentDir THEN
        _Velocity := MOVER_VELOCITY_MIN;
    ELSE
        _Velocity := -MOVER_VELOCITY_MIN;
    END_IF
END_IF

IF NOT _IsColliding AND NOT xIN_StopMover THEN

    IF DistToTravel(_CurrentPos, _TargetPos) > ABS(_Velocity) THEN
        _CurrentPos := _CurrentPos + _Velocity;

    ELSE
        _CurrentPos := _TargetPos;
        _Velocity   := 0;

    END_IF
END_IF

IF _CurrentPos >= MAX_POS THEN
    _CurrentPos := _CurrentPos - MAX_POS;
    // we prevent the stuck flag to be true at the end of the track
    THIS^._LastPos := THIS^._LastPos - MAX_POS;
END_IF

isInPos := EqualDelta(_CurrentPos, _TargetPos, 1.0); // we use delta comparison beacause axis is always at a low value 

outSimuCurrentPos   := THIS^.ResolvePos(THIS^.CurrentPos, outSimuCurrentRot);
outSimuCurrentPosSC := THIS^.ResolvePosSC(THIS^.CurrentPos, outSimuCurrentRot);

_xStuck        := (THIS^._CurrentPos < (THIS^._LastPos + _Velocity)) AND NOT isInPos;
THIS^._LastPos := THIS^._CurrentPos;

PROPERTY CurrentPos : LREAL
GET
IF CONST.BIND_WITH_TRACK THEN
    CurrentPos := TO_LREAL(gMoverAxis.I_CT_Shuttle_from_BR.asStruct[THIS^._iID].diCurrentPos_um) / 1000.0;
ELSE
    CurrentPos := _CurrentPos;
END_IF
END_GET
SET
END_SET
END_PROPERTY

PROPERTY CurrentVelocity : LREAL
GET
CurrentVelocity := THIS^._Velocity;
END_GET
SET
END_SET
END_PROPERTY

METHOD Equals : BOOL
VAR_INPUT
    object : ANY;
END_VAR
Equals := THIS = object.pValue;
END_METHOD

METHOD FB_init : BOOL
VAR_INPUT
    bInitRetains : BOOL; // if TRUE, the retain variables are initialized (warm start / cold start)
    bInCopyCode  : BOOL; // if TRUE, the instance afterwards gets moved into the copy code (online change)

    PosInit : LREAL; // initial position at startup
END_VAR
THIS^._iID := THIS^._iInstanceCounter;
THIS^._iInstanceCounter := THIS^._iInstanceCounter +1;
IF PosInit < THIS^.MAX_POS THEN
    THIS^._CurrentPos := PosInit;
ELSE
    THIS^._CurrentPos := 0;
END_IF
END_METHOD

METHOD PRIVATE GetStopLen : LREAL
VAR_INPUT
    currentVelocity : LREAL;
    currentAccel    : LREAL;
END_VAR
VAR
    tickToStop : INT;
END_VAR
// This function search the position we will get if we stop now
//
// (velocity)
//     ^          _________   <- we are here, at the end of the top slope
//     |        /          \
//     |       /            \
//     |   ___/              \______
//     |     
//     ┼------------------------------>  (time)
//
// (position)
//     ^ 
//     |                      _________
//     |                  .../
//     |               ../    ^
//     |            ../       |
//     |          ../         we search this position
//     |   ___.../
//     | 
//     ┼------------------------------>  (time)

IF currentAccel <= 0 THEN
    ASSERT(currentAccel > 0);
    RETURN;
END_IF

// TO_INT floor the result, and we need at least 1 tick to stop
tickToStop := TO_INT(currentVelocity / currentAccel) + 1;

GetStopLen := tickToStop * currentVelocity / 2;
END_METHOD

// only check the collision in one way, this prevent
// all the mover chain to be stucked
METHOD IsColliding : BOOL
VAR_INPUT
    nextMover : REFERENCE TO FB_SimuMoverAxis;
END_VAR
IsColliding := FALSE;

IF DistToTravel(THIS^.CurrentPos, nextMover.CurrentPos) <= CONST.MAX_MOVER_SIZE THEN
    IsColliding := TRUE;

END_IF

THIS^._IsColliding := IsColliding;
END_METHOD

METHOD PUBLIC MoveTo : REFERENCE TO FB_SimuMoverAxis
VAR_INPUT
    Position : LREAL; // move the axis to this position
END_VAR
THIS^._TargetPos := Position;
THIS^._CurrentDir := MoverDirection_e.Farward;
isInPos := THIS^._CurrentPos = THIS^._TargetPos;
MoveTo REF= THIS^;
END_METHOD

METHOD ResolvePos : Pos2D_t
VAR_INPUT
    inX      : LREAL;
    rotation : REFERENCE TO INT;
END_VAR
VAR CONSTANT
    (* The track has this dimension in reality
              __________
     1030mm (___________) 1030 mm
              4000 mm
			  
     and we map it like that:
	   __   80 (radius)
	  |  |
	  |  |  800
	  |  |
	  |__|
	        80 (raidus)
    *)
    START_X     : DINT  := 0;
    START_Y     : DINT  := 0;
    MAX_SIMU_DX : DINT  := 120;
    MAX_SIMU_DY : DINT  := 800;
    RADIUS_X    : LREAL := 60.0;
    RADIUS_Y    : LREAL := 100.0;

    FIRST_RADIUS_START  : LREAL := 4000;
    FIRST_RADIUS_END    : LREAL := 5030;
    SECOND_RADIUS_START : LREAL := 9030;
    SECOND_RADIUS_END   : LREAL := 10060;
END_VAR

VAR
    x_rad_calc : LREAL;
    y_rad_calc : LREAL;
    FACTOR_Y   : LREAL;
END_VAR
FACTOR_Y := FIRST_RADIUS_START / MAX_SIMU_DY;

IF inX < 0 THEN
    ResolvePos.x := START_X;
    ResolvePos.y := START_Y;
    rotation     := 0;

ELSIF inX >= 0 AND inX <= FIRST_RADIUS_START THEN
    ResolvePos.x := START_X;
    ResolvePos.y := START_Y + TO_DINT(inX / FACTOR_Y);
    rotation     := 0;

ELSIF inX > FIRST_RADIUS_START AND inX < FIRST_RADIUS_END THEN

    // should go between -1RAD and +1RAD
    x_rad_calc   := ((inX - FIRST_RADIUS_START) * 2 / (FIRST_RADIUS_END - FIRST_RADIUS_START) - 1) * PI / 2;
    ResolvePos.x := TO_DINT(SIN(x_rad_calc) * RADIUS_X) + START_X + TO_DINT(RADIUS_X);

    // should go from 0RAD to 1RAD, then 0RAD
    y_rad_calc   := (1 - (inX - FIRST_RADIUS_START) * 2 / (FIRST_RADIUS_END - FIRST_RADIUS_START)) * PI / 2;
    ResolvePos.y := TO_DINT(COS(y_rad_calc) * RADIUS_Y + START_Y + MAX_SIMU_DY);

    rotation := TO_INT(SIN(x_rad_calc) * 90 + 90);

ELSIF inX >= FIRST_RADIUS_END AND inX <= SECOND_RADIUS_START THEN
    ResolvePos.x := START_X + MAX_SIMU_DX;
    ResolvePos.y := START_Y + MAX_SIMU_DY - TO_DINT((inX - FIRST_RADIUS_END) / FACTOR_Y);
    rotation     := 180;

ELSIF inX > SECOND_RADIUS_START AND inX < SECOND_RADIUS_END THEN
    // should go between -1RAD and +1RAD
    x_rad_calc   := ((inX - SECOND_RADIUS_START) * 2 / (SECOND_RADIUS_END - SECOND_RADIUS_START) - 1) * PI / 2;
    ResolvePos.x := START_X - TO_DINT(SIN(x_rad_calc) * RADIUS_X) + TO_DINT(RADIUS_X);

    // should go from 0RAD to 1RAD, then 0RAD
    y_rad_calc   := (1 - (inX - SECOND_RADIUS_START) * 2 / (SECOND_RADIUS_END - SECOND_RADIUS_START)) * PI / 2;
    ResolvePos.y := START_Y - TO_DINT(COS(y_rad_calc) * RADIUS_Y);

    rotation := TO_INT(SIN(x_rad_calc) * 90 + 270);

ELSE
    ResolvePos.x := START_X;
    ResolvePos.y := START_Y;
    rotation     := 0;

END_IF
END_METHOD

METHOD ResolvePosSC : Pos2D_t
VAR_INPUT
    inX      : LREAL;
    rotation : REFERENCE TO INT;
END_VAR
VAR CONSTANT
    (* The track has this dimension in reality
              __________
     1030mm (___________) 1030 mm
              4000 mm
			  
     and we map it like that:
	   __   80 (radius)
	  |  |
	  |  |  800
	  |  |
	  |__|
	        80 (raidus)
    *)
    START_X     : DINT  := 0;
    START_Y     : DINT  := 0;
    MAX_SIMU_DX : DINT  := 70;
    MAX_SIMU_DY : DINT  := 800;
    RADIUS_X    : LREAL := 35;
    RADIUS_Y    : LREAL := 65.0;

    FIRST_RADIUS_START  : LREAL := 4000;
    FIRST_RADIUS_END    : LREAL := 5030;
    SECOND_RADIUS_START : LREAL := 9030;
    SECOND_RADIUS_END   : LREAL := 10060;
END_VAR

VAR
    x_rad_calc : LREAL;
    y_rad_calc : LREAL;
    FACTOR_Y   : LREAL;
END_VAR
FACTOR_Y := FIRST_RADIUS_START / MAX_SIMU_DY;

IF inX < 0 THEN
    ResolvePosSC.x := START_X;
    ResolvePosSC.y := START_Y;
    rotation       := 0;

ELSIF inX >= 0 AND inX <= FIRST_RADIUS_START THEN
    ResolvePosSC.x := START_X;
    ResolvePosSC.y := START_Y + TO_DINT(inX / FACTOR_Y);
    rotation       := 0;

ELSIF inX > FIRST_RADIUS_START AND inX < FIRST_RADIUS_END THEN

    // should go between -1RAD and +1RAD
    x_rad_calc     := ((inX - FIRST_RADIUS_START) * 2 / (FIRST_RADIUS_END - FIRST_RADIUS_START) - 1) * PI / 2;
    ResolvePosSC.x := TO_DINT(SIN(x_rad_calc) * RADIUS_X) + START_X + TO_DINT(RADIUS_X);

    // should go from 0RAD to 1RAD, then 0RAD
    y_rad_calc     := (1 - (inX - FIRST_RADIUS_START) * 2 / (FIRST_RADIUS_END - FIRST_RADIUS_START)) * PI / 2;
    ResolvePosSC.y := TO_DINT(COS(y_rad_calc) * RADIUS_Y + START_Y + MAX_SIMU_DY);

    rotation := TO_INT(SIN(x_rad_calc) * 90 + 90);

ELSIF inX >= FIRST_RADIUS_END AND inX <= SECOND_RADIUS_START THEN
    ResolvePosSC.x := START_X + MAX_SIMU_DX;
    ResolvePosSC.y := START_Y + MAX_SIMU_DY - TO_DINT((inX - FIRST_RADIUS_END) / FACTOR_Y);
    rotation       := 180;

ELSIF inX > SECOND_RADIUS_START AND inX < SECOND_RADIUS_END THEN
    // should go between -1RAD and +1RAD
    x_rad_calc     := ((inX - SECOND_RADIUS_START) * 2 / (SECOND_RADIUS_END - SECOND_RADIUS_START) - 1) * PI / 2;
    ResolvePosSC.x := START_X - TO_DINT(SIN(x_rad_calc) * RADIUS_X) + TO_DINT(RADIUS_X);

    // should go from 0RAD to 1RAD, then 0RAD
    y_rad_calc     := (1 - (inX - SECOND_RADIUS_START) * 2 / (SECOND_RADIUS_END - SECOND_RADIUS_START)) * PI / 2;
    ResolvePosSC.y := START_Y - TO_DINT(COS(y_rad_calc) * RADIUS_Y);

    rotation := TO_INT(SIN(x_rad_calc) * 90 + 270);

ELSE
    ResolvePosSC.x := START_X;
    ResolvePosSC.y := START_Y;
    rotation       := 0;

END_IF

ResolvePosSC.x := -ResolvePosSC.x;
END_METHOD

METHOD ToString : STRING
VAR_INPUT
END_VAR
VAR
END_VAR
ToString := CONCAT('FB_SimuMoverAxis_', TO_STRING(THIS^._iID));
END_METHOD

// Use this method in a collider manager so the simu axis 
// will know when to stop itself
METHOD WillCollide : BOOL
VAR_INPUT
    nextMover : REFERENCE TO FB_SimuMoverAxis;
END_VAR
VAR
    diffVelocity : LREAL;
END_VAR
THIS^._willCollide := FALSE;
diffVelocity       := 0;

// If the 2 movers are moving tarwards each other
IF (THIS^._Velocity > 0) AND (nextMover.CurrentVelocity < 0) THEN
    diffVelocity := SQRT(THIS^._Velocity * THIS^._Velocity + (nextMover.CurrentVelocity * nextMover.CurrentVelocity));

    // If the 2 movers are moving in the same direction
ELSE
    IF ABS(THIS^._Velocity) > ABS(nextMover.CurrentVelocity) THEN
        diffVelocity :=
            SQRT(THIS^._Velocity * THIS^._Velocity - (nextMover.CurrentVelocity * nextMover.CurrentVelocity));
    END_IF
END_IF

THIS^._willCollide
    := DistToTravel(THIS^.CurrentPos, nextMover.CurrentPos) <=
       THIS^.GetStopLen(diffVelocity, SIMU.lrAccelMover) + CONST.MAX_MOVER_SIZE;

WillCollide := THIS^._willCollide;
END_METHOD

PROPERTY xStuck : BOOL
GET
xStuck := _xStuck;
END_GET
SET
END_SET
END_PROPERTY

END_FUNCTION_BLOCK

// ---- POUs/20_AUTO/Mover/DistToTravel.TcPOU
// Get the distance to travel from startPos to stopPos
FUNCTION DistToTravel : LREAL
VAR_INPUT
    startPos : LREAL;
    stopPos  : LREAL;
END_VAR
VAR
END_VAR

IF startPos > stopPos THEN
    DistToTravel := stopPos - startPos + CONST.MAX_TRACK_LENGTH;
ELSE
    DistToTravel := stopPos - startPos;
END_IF

END_FUNCTION

// ---- POUs/20_AUTO/TOOL/EqualDelta.TcPOU
// Check if 2 lreal positions are equal, using a delta method
// Please be sure that a and b stays aroud 0 because this function
// depend on your floating point accuracy !
// Always prefer IsPosEqualEpsilon when possible
FUNCTION EqualDelta : BOOL
VAR_INPUT
    a     : LREAL; // first pos
    b     : LREAL; // second pos
    delta : LREAL; // if position is between ]+/-[ delta (not included) then return true
END_VAR
VAR
END_VAR

EqualDelta := (b < a+delta) AND (b>a-delta);

END_FUNCTION

// ---- POUs/20_AUTO/TOOL/ASSERT.TcPOU
FUNCTION ASSERT : BOOL
VAR_INPUT
    bStatement : BOOL; // Should be true, else raise an error
END_VAR
VAR
END_VAR

IF NOT  bStatement THEN
	{error <'Assertion has occured'>}
	ASSERT := TRUE;
ELSE
	ASSERT := FALSE;
END_IF

END_FUNCTION

// ---- POUs/20_AUTO/Mover/FB_Mover.TcPOU
FUNCTION_BLOCK FB_Mover IMPLEMENTS IObject
VAR_INPUT
END_VAR
VAR_OUTPUT
END_VAR
VAR
    _ID           : INT;                           // hard id number of the mover
    _MoverAxis    : REFERENCE TO FB_SimuMoverAxis; // reference to an FB_SimuMoverAxis
    _AttachedTool : ARRAY [0..3] OF FB_PieceHolderMover(0,0,0,0);   // attached toolhead
    _Station      : REFERENCE TO FB_Station;       // current station

    _State : MoverState_e := MoverState_e.WaitOnNextStation; // current mover state

    _ActualTargetOffset  : LREAL; // final offset to apply to the current/next target
    _MovingProcessOffset : LREAL; (* added offset by the process, 
                                     used to compute the new position of the shuttle inside the station *)

    _iID : INT := 0; // instance ID, is set during FB_Init using the value of _iInstanceCounter 
END_VAR
VAR CONSTANT
END_VAR
VAR_STAT
    _iInstanceCounter : INT := 1; // instance counter
END_VAR

// Abort all current actions and go to the given station
METHOD PUBLIC Abort : BOOL
VAR_INPUT
	Station : REFERENCE TO FB_Station;
END_VAR
THIS^.State := MoverState_e.OperationDone;

IF __ISVALIDREF(THIS^.Station) AND_THEN __ISVALIDREF(THIS^.Station.Process) THEN
    THIS^.Station.Process.TakeMover();
END_IF

IF __ISVALIDREF(Station) THEN
    THIS^.SetStation(Station);
    THIS^.MoveToStation();
    THIS^.State := MoverState_e.MovingToStation;
END_IF
END_METHOD

// This is the final offset to apply when moving to a target
PROPERTY PUBLIC ActualTargetOffset : LREAL
GET
ActualTargetOffset := THIS^._ActualTargetOffset;
END_GET
END_PROPERTY

METHOD Equals : BOOL
VAR_INPUT
    object : ANY;
END_VAR
Equals := THIS = object.pValue;
END_METHOD

METHOD FB_init : BOOL
VAR_INPUT
    bInitRetains : BOOL; // if TRUE, the retain variables are initialized (warm start / cold start)
    bInCopyCode  : BOOL; // if TRUE, the instance afterwards gets moved into the copy code (online change)
    ID           : INT;  // hard id number of the mover

    MoverAxis : REFERENCE TO FB_SimuMoverAxis; // reference to an FB_SimuMoverAxis
END_VAR
THIS^._iID := THIS^._iInstanceCounter;
THIS^._iInstanceCounter := THIS^._iInstanceCounter +1;
THIS^._ID := ID;
THIS^._MoverAxis REF= MoverAxis;
THIS^._Station REF=0;
END_METHOD

METHOD PUBLIC GetPiece : REFERENCE TO FB_My_Piece
VAR_INPUT
    PieceLocation : PiecePos_e;
END_VAR
IF PieceLocation >= 0 AND PieceLocation < PiecePos_e._max THEN
    GetPiece REF= THIS^._AttachedTool[PieceLocation].GetPiece();
END_IF
END_METHOD

// Is this mover behind a given position?
// this method do the opposit as IsInFront
METHOD IsBehind : BOOL
VAR_INPUT
    lrPosition : LREAL; // position to test
END_VAR
IsBehind := lrPosition > THIS^._MoverAxis.CurrentPos;
END_METHOD

// Is this mover is in front of a given position?
// Use this function also to check if the next station is behind the mover or not.
// In this case, the mover needs to complet its turn for accessing the given station
METHOD IsInFront : BOOL
VAR_INPUT
    lrPosition : LREAL; // position to test
END_VAR
IsInFront := lrPosition < THIS^._MoverAxis.CurrentPos;
END_METHOD

METHOD IsInStationPos : BOOL
VAR_INPUT
END_VAR
// we have to substract the piecholder offset to find the station position again
IF CONST.BIND_WITH_TRACK THEN
    // IsInStationPos :=
    //     THIS^.Station.Position.isInPos(gMoverAxis.I_CT_Shuttle_from_BR.asStruct[THIS^._ID].diCurrentPos_um / 1000 -
    //                                    THIS^._AttachedTool[0].PosOffset -
    //                                    THIS^.Station.Offset);
    IF __ISVALIDREF(THIS^.Station) THEN
        //IsInStationPos :=
        //    gMoverAxis.I_CT_Shuttle_from_BR.asStruct[THIS^._ID].bStatus.at_target AND
        //    (gMoverAxis.I_CT_Shuttle_from_BR.asStruct[THIS^._ID].bDestinationStation = THIS^.Station.SuperTrackNumber);
        IsInStationPos :=
            THIS^.Station.Position.isInPos(gMoverAxis.I_CT_Shuttle_from_BR.asStruct[THIS^._ID].diCurrentPos_um / 1000 -
                                           THIS^._AttachedTool[0].PosOffset -
                                           THIS^.Station.Offset -
                                           THIS^._MovingProcessOffset) AND
            gMoverAxis.I_CT_Shuttle_from_BR.asStruct[THIS^._ID].bStatus.at_target;
    ELSE
        IsInStationPos := FALSE;
    END_IF
ELSE
    IsInStationPos := THIS^.Station.Position.isInPos(THIS^.MoverAxis.CurrentPos -
                                                     THIS^._AttachedTool[0].PosOffset -
                                                     THIS^.Station.Offset -
                                                     THIS^._MovingProcessOffset);
END_IF
END_METHOD

PROPERTY MoverAxis : REFERENCE TO FB_SimuMoverAxis
GET
MoverAxis REF= _MoverAxis;
END_GET
SET
_MoverAxis REF= MoverAxis;
END_SET
END_PROPERTY

// When a mover is given to a process, this process is allowed to
// use this command to move the shuttle
METHOD PUBLIC MoveRelativeInsideStation : BOOL
VAR_INPUT
    offsetPosition : LREAL;
END_VAR
MoveRelativeInsideStation := FALSE;

IF (MoverState_e.InOperation = THIS^.State) AND
   (ABS(offsetPosition + THIS^.Station.Offset + THIS^._MovingProcessOffset) < LREAL#500.0) THEN
    THIS^.State                := MoverState_e.PerformRelativeMove;
    THIS^._MovingProcessOffset := offsetPosition + THIS^._MovingProcessOffset;
    THIS^.MoverAxis.MoveTo(TO_POS(THIS^.Station.Position.lrWorkPosition +
                                  THIS^._AttachedTool[0].PosOffset +
                                  THIS^.Station.Offset +
                                  THIS^._MovingProcessOffset));

    MoveRelativeInsideStation := TRUE;
END_IF
END_METHOD

// Move to the current set station. Can only move if the current process are running
METHOD MoveToStation : REFERENCE TO FB_Mover
VAR_INPUT
END_VAR
IF THIS^._State <> MoverState_e.InOperation THEN
    THIS^.MoverAxis
        .MoveTo(TO_POS(THIS^.Station.Position.lrWorkPosition + THIS^._AttachedTool[0].PosOffset + THIS^.Station.Offset));

    THIS^._MovingProcessOffset := 0;
    THIS^._ActualTargetOffset  := THIS^._AttachedTool[0].PosOffset + THIS^.Station.Offset;
    THIS^._State               := MoverState_e.WaitLeaveCurrentStation;
ELSE
    ASSERT(0); // should not be called when we are in operation !
END_IF

MoveToStation REF= THIS^;
END_METHOD

// Move to waiting spot
// The mover will not move if the waiting spot can not store
// a full mover
METHOD MoveToWaitSpot : REFERENCE TO FB_Mover
VAR_INPUT
END_VAR
IF THIS^._State <> MoverState_e.InOperation THEN
    IF THIS^.Station.WaitPos <= (THIS^.Station.Position.lrWorkPosition - CONST.MAX_MOVER_SIZE) THEN
        THIS^.MoverAxis.MoveTo(TO_POS(THIS^.Station.WaitPos + THIS^._AttachedTool[0].PosOffset + THIS^.Station.Offset));
    ELSE
        THIS^.MoverAxis.MoveTo(TO_POS(THIS^.Station.Position.lrWorkPosition +
                                      THIS^._AttachedTool[0].PosOffset +
                                      THIS^.Station.Offset));
    END_IF

    THIS^._MovingProcessOffset := 0;
    THIS^._ActualTargetOffset  := THIS^._AttachedTool[0].PosOffset + THIS^.Station.Offset + THIS^.Station._WaitPosOffset;
    THIS^._State               := MoverState_e.WaitLeaveCurrentStation;
ELSE
    ASSERT(0); // never use this command when we are in operation
END_IF

MoveToWaitSpot REF= THIS^;
END_METHOD

PROPERTY PUBLIC MovingProcessOffset : LREAL
GET
MovingProcessOffset := THIS^._MovingProcessOffset;
END_GET
END_PROPERTY

// Set a specic piece holder. This will affect the station position offset
METHOD SetPieceHolder : REFERENCE TO FB_Mover
VAR_INPUT
	pieceHolder : REFERENCE TO FB_PieceHolderMover;
END_VAR
// do nothing
SetPieceHolder REF= THIS^;
END_METHOD

// Set the next station of the mover. This action does not make the mover moves. 
// First you need to set the station. Then, depending on the station scenario,
// you will run to it when its current process is finished or move to it
// as quick as possible
METHOD SetStation : REFERENCE TO FB_Mover
VAR_INPUT
	Station : REFERENCE TO FB_Station;
END_VAR
IF __ISVALIDREF(Station) AND_THEN (THIS^._State <> MoverState_e.InOperation) THEN
    THIS^._Station REF= Station;
    THIS^._State   := MoverState_e.WaitOnNextStation;
ELSE
    ASSERT(0);
END_IF

SetStation REF= THIS^;
END_METHOD

PROPERTY State : MoverState_e
GET
State := _State;
END_GET
SET
_State := State;
END_SET
END_PROPERTY

PROPERTY Station : REFERENCE TO FB_Station
GET
Station REF=_Station;
END_GET
SET
_Station REF=Station;
END_SET
END_PROPERTY

